LIN {X 0.120,Y -301.447,Z 452.705,A 0.000,B 0.000,C 90.000,E1 126.870} C_DIS
LIN {X -0.059,Y -305.207,Z 452.702,A 0.000,B 0.000,C 90.000,E1 126.423} C_DIS
LIN {X -0.045,Y -307.018,Z 452.700,A 0.000,B 0.000,C 90.000,E1 126.091} C_DIS
LIN {X 0.151,Y -308.441,Z 452.699,A 0.000,B 0.000,C 90.000,E1 125.724} C_DIS
LIN {X 0.025,Y -313.580,Z 452.690,A 0.000,B 0.000,C 90.000,E1 124.119} C_DIS
LIN {X 0.115,Y -323.537,Z 452.673,A 0.000,B 0.000,C 90.000,E1 121.209} C_DIS
LIN {X 0.173,Y -334.816,Z 452.658,A 0.000,B 0.000,C 90.000,E1 118.359} C_DIS
LIN {X 0.070,Y -347.524,Z 452.642,A 0.000,B 0.000,C 90.000,E1 115.591} C_DIS
LIN {X -0.180,Y -360.110,Z 452.629,A 0.000,B 0.000,C 90.000,E1 113.206} C_DIS
LIN {X 0.078,Y -374.006,Z 452.616,A 0.000,B 0.000,C 90.000,E1 110.791} C_DIS
LIN {X -0.054,Y -389.312,Z 452.603,A 0.000,B 0.000,C 90.000,E1 108.489} C_DIS
LIN {X 0.080,Y -406.143,Z 452.590,A 0.000,B 0.000,C 90.000,E1 106.205} C_DIS
LIN {X 0.012,Y -424.621,Z 452.578,A 0.000,B 0.000,C 90.000,E1 104.008} C_DIS
LIN {X 0.142,Y -444.522,Z 452.566,A 0.000,B 0.000,C 90.000,E1 101.883} C_DIS
LIN {X 0.031,Y -465.029,Z 452.555,A 0.000,B 0.000,C 90.000,E1 99.962} C_DIS
LIN {X 0.056,Y -483.349,Z 452.547,A 0.000,B 0.000,C 90.000,E1 98.398} C_DIS
LIN {X 0.226,Y -485.471,Z 452.546,A 0.000,B 0.000,C 90.000,E1 98.163} C_DIS
LIN {X 0.064,Y -487.300,Z 452.544,A 0.000,B 0.000,C 90.000,E1 97.936} C_DIS
LIN {X -0.032,Y -488.676,Z 452.543,A 0.000,B 0.000,C 90.000,E1 97.701} C_DIS
LIN {X 0.176,Y -490.427,Z 452.540,A 0.000,B 0.000,C 90.000,E1 97.182} C_DIS
LIN {X -0.095,Y -491.085,Z 452.537,A 0.000,B 0.000,C 90.000,E1 96.720} C_DIS
LIN {X 0.132,Y -490.756,Z 452.535,A 0.000,B 0.000,C 90.000,E1 96.201} C_DIS
LIN {X -0.126,Y -489.389,Z 452.532,A 0.000,B 0.000,C 90.000,E1 95.739} C_DIS
LIN {X 0.208,Y -488.246,Z 452.530,A 0.000,B 0.000,C 90.000,E1 95.454} C_DIS
LIN {X 0.100,Y -486.714,Z 452.529,A 0.000,B 0.000,C 90.000,E1 95.220} C_DIS
LIN {X -0.023,Y -478.801,Z 452.524,A 0.000,B 0.000,C 90.000,E1 94.245} C_DIS
LIN {X -0.206,Y -457.268,Z 452.508,A 0.000,B 0.000,C 90.000,E1 91.489} C_DIS
LIN {X -0.024,Y -444.971,Z 452.498,A 0.000,B 0.000,C 90.000,E1 89.656} C_DIS
LIN {X -0.084,Y -433.386,Z 452.488,A 0.000,B 0.000,C 90.000,E1 87.822} C_DIS
LIN {X -0.117,Y -418.721,Z 452.474,A 0.000,B 0.000,C 90.000,E1 85.412} C_DIS
LIN {X -0.119,Y -406.257,Z 452.462,A 0.000,B 0.000,C 90.000,E1 83.223} C_DIS
LIN {X 0.015,Y -395.531,Z 452.451,A 0.000,B 0.000,C 90.000,E1 81.254} C_DIS
LIN {X -0.039,Y -383.227,Z 452.439,A 0.000,B 0.000,C 90.000,E1 78.993} C_DIS
LIN {X -0.169,Y -368.243,Z 452.423,A 0.000,B 0.000,C 90.000,E1 76.117} C_DIS
LIN {X -0.106,Y -356.985,Z 452.410,A 0.000,B 0.000,C 90.000,E1 73.740} C_DIS
LIN {X -0.151,Y -342.943,Z 452.391,A 0.000,B 0.000,C 90.000,E1 70.423} C_DIS
LIN {X 0.038,Y -332.368,Z 452.376,A 0.000,B 0.000,C 90.000,E1 67.614} C_DIS
LIN {X 0.001,Y -321.989,Z 452.360,A 0.000,B 0.000,C 90.000,E1 64.793} C_DIS
LIN {X 0.035,Y -313.043,Z 452.346,A 0.000,B 0.000,C 90.000,E1 62.231} C_DIS
LIN {X -0.129,Y -304.242,Z 452.331,A 0.000,B 0.000,C 90.000,E1 59.665} C_DIS
LIN {X 0.016,Y -293.773,Z 452.313,A 0.000,B 0.000,C 90.000,E1 56.342} C_DIS
LIN {X 0.083,Y -284.083,Z 452.294,A 0.000,B 0.000,C 90.000,E1 52.970} C_DIS
LIN {X -0.107,Y -278.413,Z 452.283,A 0.000,B 0.000,C 90.000,E1 50.964} C_DIS
LIN {X 0.119,Y -272.507,Z 452.272,A 0.000,B 0.000,C 90.000,E1 48.852} C_DIS
LIN {X 0.026,Y -266.367,Z 452.260,A 0.000,B 0.000,C 90.000,E1 46.782} C_DIS
LIN {X -0.007,Y -260.067,Z 452.248,A 0.000,B 0.000,C 90.000,E1 44.676} C_DIS
LIN {X 0.030,Y -253.666,Z 452.236,A 0.000,B 0.000,C 90.000,E1 42.528} C_DIS
LIN {X -0.018,Y -245.018,Z 452.220,A 0.000,B 0.000,C 90.000,E1 39.644} C_DIS
LIN {X 0.084,Y -234.685,Z 452.200,A 0.000,B 0.000,C 90.000,E1 35.931} C_DIS
LIN {X -0.057,Y -227.197,Z 452.183,A 0.000,B 0.000,C 90.000,E1 32.959} C_DIS
LIN {X 0.072,Y -220.483,Z 452.166,A 0.000,B 0.000,C 90.000,E1 29.873} C_DIS
LIN {X 0.003,Y -214.671,Z 452.149,A 0.000,B 0.000,C 90.000,E1 26.796} C_DIS
LIN {X -0.085,Y -208.369,Z 452.127,A 0.000,B 0.000,C 90.000,E1 22.898} C_DIS
LIN {X -0.020,Y -203.087,Z 452.105,A 0.000,B 0.000,C 90.000,E1 18.906} C_DIS
LIN {X -0.056,Y -198.758,Z 452.083,A 0.000,B 0.000,C 90.000,E1 14.898} C_DIS
LIN {X -0.018,Y -194.835,Z 452.056,A 0.000,B 0.000,C 90.000,E1 10.018} C_DIS
LIN {X -0.064,Y -191.927,Z 452.024,A 0.000,B 0.000,C 90.000,E1 4.302} C_DIS
LIN {X 0.083,Y -191.956,Z 451.965,A 0.000,B 0.000,C 90.000,E1 353.742} C_DIS
LIN {X 0.097,Y -194.918,Z 451.933,A 0.000,B 0.000,C 90.000,E1 347.993} C_DIS
LIN {X -0.034,Y -198.884,Z 451.906,A 0.000,B 0.000,C 90.000,E1 343.142} C_DIS
LIN {X 0.035,Y -203.206,Z 451.884,A 0.000,B 0.000,C 90.000,E1 339.082} C_DIS
LIN {X -0.034,Y -208.624,Z 451.862,A 0.000,B 0.000,C 90.000,E1 335.101} C_DIS
LIN {X 0.041,Y -214.800,Z 451.840,A 0.000,B 0.000,C 90.000,E1 331.129} C_DIS
LIN {X -0.027,Y -221.542,Z 451.818,A 0.000,B 0.000,C 90.000,E1 327.248} C_DIS
LIN {X -0.075,Y -228.974,Z 451.797,A 0.000,B 0.000,C 90.000,E1 323.417} C_DIS
LIN {X -0.031,Y -237.180,Z 451.776,A 0.000,B 0.000,C 90.000,E1 319.622} C_DIS
LIN {X 0.023,Y -246.445,Z 451.755,A 0.000,B 0.000,C 90.000,E1 315.891} C_DIS
LIN {X 0.032,Y -256.044,Z 451.737,A 0.000,B 0.000,C 90.000,E1 312.609} C_DIS
LIN {X 0.055,Y -268.123,Z 451.717,A 0.000,B 0.000,C 90.000,E1 309.036} C_DIS
LIN {X 0.111,Y -280.070,Z 451.699,A 0.000,B 0.000,C 90.000,E1 305.884} C_DIS
LIN {X 0.018,Y -294.154,Z 451.681,A 0.000,B 0.000,C 90.000,E1 302.498} C_DIS
LIN {X -0.144,Y -307.643,Z 451.664,A 0.000,B 0.000,C 90.000,E1 299.539} C_DIS
LIN {X -0.045,Y -320.638,Z 451.650,A 0.000,B 0.000,C 90.000,E1 296.924} C_DIS
LIN {X -0.046,Y -334.871,Z 451.635,A 0.000,B 0.000,C 90.000,E1 294.387} C_DIS
LIN {X 0.021,Y -346.380,Z 451.625,A 0.000,B 0.000,C 90.000,E1 292.514} C_DIS
LIN {X -0.181,Y -363.228,Z 451.612,A 0.000,B 0.000,C 90.000,E1 290.120} C_DIS
LIN {X 0.035,Y -386.462,Z 451.595,A 0.000,B 0.000,C 90.000,E1 287.149} C_DIS
LIN {X -0.172,Y -401.479,Z 451.586,A 0.000,B 0.000,C 90.000,E1 285.481} C_DIS
LIN {X 0.187,Y -424.373,Z 451.573,A 0.000,B 0.000,C 90.000,E1 283.119} C_DIS
LIN {X 0.111,Y -434.478,Z 451.567,A 0.000,B 0.000,C 90.000,E1 282.119} C_DIS
LIN {X -0.239,Y -444.292,Z 451.562,A 0.000,B 0.000,C 90.000,E1 281.130} C_DIS
LIN {X 0.076,Y -451.255,Z 451.557,A 0.000,B 0.000,C 90.000,E1 280.310} C_DIS
LIN {X -0.146,Y -457.806,Z 451.553,A 0.000,B 0.000,C 90.000,E1 279.557} C_DIS
LIN {X 0.151,Y -463.921,Z 451.549,A 0.000,B 0.000,C 90.000,E1 278.746} C_DIS
LIN {X 0.043,Y -469.402,Z 451.544,A 0.000,B 0.000,C 90.000,E1 277.992} C_DIS
LIN {X -0.017,Y -474.376,Z 451.540,A 0.000,B 0.000,C 90.000,E1 277.239} C_DIS
LIN {X -0.234,Y -480.245,Z 451.535,A 0.000,B 0.000,C 90.000,E1 276.258} C_DIS
LIN {X -0.261,Y -484.098,Z 451.530,A 0.000,B 0.000,C 90.000,E1 275.511} C_DIS
LIN {X -0.080,Y -486.395,Z 451.528,A 0.000,B 0.000,C 90.000,E1 274.992} C_DIS
LIN {X 0.114,Y -488.309,Z 451.525,A 0.000,B 0.000,C 90.000,E1 274.473} C_DIS
LIN {X -0.176,Y -489.851,Z 451.522,A 0.000,B 0.000,C 90.000,E1 274.012} C_DIS
LIN {X 0.001,Y -490.957,Z 451.519,A 0.000,B 0.000,C 90.000,E1 273.498} C_DIS
LIN {X 0.216,Y -491.675,Z 451.517,A 0.000,B 0.000,C 90.000,E1 272.980} C_DIS
LIN {X -0.079,Y -492.019,Z 451.514,A 0.000,B 0.000,C 90.000,E1 272.522} C_DIS
LIN {X 0.125,Y -491.944,Z 451.511,A 0.000,B 0.000,C 90.000,E1 272.007} C_DIS
LIN {X -0.144,Y -491.479,Z 451.508,A 0.000,B 0.000,C 90.000,E1 271.547} C_DIS
LIN {X 0.060,Y -490.612,Z 451.506,A 0.000,B 0.000,C 90.000,E1 271.031} C_DIS
LIN {X -0.225,Y -489.255,Z 451.503,A 0.000,B 0.000,C 90.000,E1 270.573} C_DIS
LIN {X -0.026,Y -487.379,Z 451.500,A 0.000,B 0.000,C 90.000,E1 270.057} C_DIS
LIN {X 0.164,Y -484.887,Z 451.498,A 0.000,B 0.000,C 90.000,E1 269.542} C_DIS
LIN {X -0.148,Y -481.651,Z 451.495,A 0.000,B 0.000,C 90.000,E1 269.083} C_DIS
LIN {X 0.005,Y -477.481,Z 451.492,A 0.000,B 0.000,C 90.000,E1 268.568} C_DIS
LIN {X -0.167,Y -475.019,Z 451.491,A 0.000,B 0.000,C 90.000,E1 268.339} C_DIS
LIN {X 0.129,Y -469.421,Z 451.488,A 0.000,B 0.000,C 90.000,E1 267.822} C_DIS
LIN {X -0.119,Y -463.170,Z 451.486,A 0.000,B 0.000,C 90.000,E1 267.421} C_DIS
LIN {X 0.143,Y -456.577,Z 451.484,A 0.000,B 0.000,C 90.000,E1 267.020} C_DIS
LIN {X -0.034,Y -449.739,Z 451.482,A 0.000,B 0.000,C 90.000,E1 266.731} C_DIS
LIN {X 0.132,Y -442.560,Z 451.480,A 0.000,B 0.000,C 90.000,E1 266.445} C_DIS
LIN {X -0.190,Y -434.851,Z 451.479,A 0.000,B 0.000,C 90.000,E1 266.274} C_DIS
LIN {X -0.091,Y -426.271,Z 451.478,A 0.000,B 0.000,C 90.000,E1 266.102} C_DIS
LIN {X -0.040,Y -414.893,Z 451.478,A 0.000,B 0.000,C 90.000,E1 265.988} C_DIS
LIN {X 0.146,Y -408.689,Z 451.478,A 0.000,B 0.000,C 90.000,E1 265.931} C_DIS
LIN {X 0.044,Y -180.918,Z 451.477,A 0.000,B 0.000,C 90.000,E1 265.927} C_DIS
LIN {X 0.076,Y -180.841,Z 451.472,A 0.000,B 0.000,C 90.000,E1 264.894} C_DIS
LIN {X -0.027,Y -178.883,Z 451.443,A 0.000,B 0.000,C 90.000,E1 259.690} C_DIS
LIN {X 0.048,Y -175.926,Z 451.414,A 0.000,B 0.000,C 90.000,E1 254.574} C_DIS
LIN {X -0.006,Y -175.365,Z 451.410,A 0.000,B 0.000,C 90.000,E1 253.740} C_DIS
LIN {X 0.052,Y -172.143,Z 451.386,A 0.000,B 0.000,C 90.000,E1 249.444} C_DIS
LIN {X 0.029,Y -171.608,Z 451.381,A 0.000,B 0.000,C 90.000,E1 248.592} C_DIS
LIN {X 0.018,Y -167.830,Z 451.357,A 0.000,B 0.000,C 90.000,E1 244.280} C_DIS
LIN {X 0.035,Y -166.556,Z 451.348,A 0.000,B 0.000,C 90.000,E1 242.538} C_DIS
LIN {X -0.054,Y -162.551,Z 451.323,A 0.000,B 0.000,C 90.000,E1 238.201} C_DIS
LIN {X 0.005,Y -161.229,Z 451.313,A 0.000,B 0.000,C 90.000,E1 236.421} C_DIS
LIN {X 0.041,Y -157.234,Z 451.289,A 0.000,B 0.000,C 90.000,E1 231.984} C_DIS
LIN {X 0.064,Y -155.959,Z 451.279,A 0.000,B 0.000,C 90.000,E1 230.194} C_DIS
LIN {X 0.021,Y -152.213,Z 451.254,A 0.000,B 0.000,C 90.000,E1 225.729} C_DIS
LIN {X 0.042,Y -150.457,Z 451.239,A 0.000,B 0.000,C 90.000,E1 223.014} C_DIS
LIN {X 0.069,Y -147.183,Z 451.214,A 0.000,B 0.000,C 90.000,E1 218.463} C_DIS
LIN {X 0.035,Y -145.201,Z 451.194,A 0.000,B 0.000,C 90.000,E1 214.818} C_DIS
LIN {X -0.055,Y -142.338,Z 451.163,A 0.000,B 0.000,C 90.000,E1 209.333} C_DIS
LIN {X -0.001,Y -141.727,Z 451.153,A 0.000,B 0.000,C 90.000,E1 207.462} C_DIS
LIN {X -0.019,Y -139.480,Z 451.116,A 0.000,B 0.000,C 90.000,E1 200.972} C_DIS
LIN {X -0.030,Y -138.979,Z 451.101,A 0.000,B 0.000,C 90.000,E1 198.181} C_DIS
LIN {X -0.045,Y -138.332,Z 451.054,A 0.000,B 0.000,C 90.000,E1 189.782} C_DIS
LIN {X -0.045,Y -139.429,Z 451.008,A 0.000,B 0.000,C 90.000,E1 181.375} C_DIS
LIN {X 0.008,Y -141.357,Z 450.971,A 0.000,B 0.000,C 90.000,E1 174.837} C_DIS
LIN {X -0.016,Y -142.711,Z 450.956,A 0.000,B 0.000,C 90.000,E1 172.064} C_DIS
LIN {X -0.056,Y -145.086,Z 450.930,A 0.000,B 0.000,C 90.000,E1 167.465} C_DIS
LIN {X -0.061,Y -147.710,Z 450.910,A 0.000,B 0.000,C 90.000,E1 163.795} C_DIS
LIN {X 0.022,Y -150.365,Z 450.890,A 0.000,B 0.000,C 90.000,E1 160.115} C_DIS
LIN {X 0.041,Y -153.792,Z 450.869,A 0.000,B 0.000,C 90.000,E1 156.485} C_DIS
LIN {X -0.039,Y -157.204,Z 450.849,A 0.000,B 0.000,C 90.000,E1 152.922} C_DIS
LIN {X 0.042,Y -161.366,Z 450.830,A 0.000,B 0.000,C 90.000,E1 149.331} C_DIS
LIN {X 0.053,Y -165.569,Z 450.810,A 0.000,B 0.000,C 90.000,E1 145.801} C_DIS
LIN {X -0.063,Y -170.486,Z 450.791,A 0.000,B 0.000,C 90.000,E1 142.351} C_DIS
LIN {X 0.086,Y -175.368,Z 450.772,A 0.000,B 0.000,C 90.000,E1 138.852} C_DIS
LIN {X -0.051,Y -180.991,Z 450.753,A 0.000,B 0.000,C 90.000,E1 135.486} C_DIS
LIN {X 0.073,Y -186.418,Z 450.734,A 0.000,B 0.000,C 90.000,E1 132.081} C_DIS
LIN {X -0.126,Y -191.046,Z 450.720,A 0.000,B 0.000,C 90.000,E1 129.644} C_DIS
LIN {X 0.003,Y -195.023,Z 450.707,A 0.000,B 0.000,C 90.000,E1 127.282} C_DIS
LIN {X -0.030,Y -292.656,Z 450.707,A 0.000,B 0.000,C 90.000,E1 127.282} C_DIS
LIN {X -0.113,Y -297.600,Z 450.706,A 0.000,B 0.000,C 90.000,E1 127.156} C_DIS
LIN {X 0.008,Y -300.299,Z 450.705,A 0.000,B 0.000,C 90.000,E1 126.950} C_DIS
LIN {X 0.027,Y -304.083,Z 450.703,A 0.000,B 0.000,C 90.000,E1 126.537} C_DIS
LIN {X 0.135,Y -306.022,Z 450.701,A 0.000,B 0.000,C 90.000,E1 126.217} C_DIS
LIN {X 0.059,Y -307.557,Z 450.700,A 0.000,B 0.000,C 90.000,E1 125.931} C_DIS
LIN {X 0.090,Y -308.890,Z 450.698,A 0.000,B 0.000,C 90.000,E1 125.598} C_DIS
LIN {X -0.005,Y -320.535,Z 450.678,A 0.000,B 0.000,C 90.000,E1 122.054} C_DIS
LIN {X -0.048,Y -331.424,Z 450.662,A 0.000,B 0.000,C 90.000,E1 119.205} C_DIS
LIN {X -0.103,Y -343.712,Z 450.647,A 0.000,B 0.000,C 90.000,E1 116.411} C_DIS
LIN {X 0.013,Y -355.896,Z 450.633,A 0.000,B 0.000,C 90.000,E1 113.951} C_DIS
LIN {X 0.168,Y -369.359,Z 450.620,A 0.000,B 0.000,C 90.000,E1 111.535} C_DIS
LIN {X 0.055,Y -384.199,Z 450.607,A 0.000,B 0.000,C 90.000,E1 109.214} C_DIS
LIN {X 0.181,Y -400.526,Z 450.594,A 0.000,B 0.000,C 90.000,E1 106.913} C_DIS
LIN {X -0.028,Y -418.459,Z 450.582,A 0.000,B 0.000,C 90.000,E1 104.717} C_DIS
LIN {X 0.194,Y -438.015,Z 450.570,A 0.000,B 0.000,C 90.000,E1 102.535} C_DIS
LIN {X 0.191,Y -458.346,Z 450.559,A 0.000,B 0.000,C 90.000,E1 100.546} C_DIS
LIN {X -0.250,Y -484.346,Z 450.546,A 0.000,B 0.000,C 90.000,E1 98.341} C_DIS
LIN {X -0.039,Y -487.846,Z 450.544,A 0.000,B 0.000,C 90.000,E1 97.871} C_DIS
LIN {X -0.220,Y -489.138,Z 450.542,A 0.000,B 0.000,C 90.000,E1 97.644} C_DIS
LIN {X 0.150,Y -490.088,Z 450.541,A 0.000,B 0.000,C 90.000,E1 97.352} C_DIS
LIN {X -0.120,Y -491.128,Z 450.538,A 0.000,B 0.000,C 90.000,E1 96.891} C_DIS
LIN {X 0.103,Y -491.164,Z 450.535,A 0.000,B 0.000,C 90.000,E1 96.372} C_DIS
LIN {X -0.155,Y -490.200,Z 450.533,A 0.000,B 0.000,C 90.000,E1 95.910} C_DIS
LIN {X 0.072,Y -488.065,Z 450.530,A 0.000,B 0.000,C 90.000,E1 95.391} C_DIS
LIN {X -0.082,Y -486.413,Z 450.529,A 0.000,B 0.000,C 90.000,E1 95.163} C_DIS
LIN {X 0.137,Y -476.456,Z 450.522,A 0.000,B 0.000,C 90.000,E1 93.898} C_DIS
LIN {X 0.076,Y -456.937,Z 450.508,A 0.000,B 0.000,C 90.000,E1 91.375} C_DIS
LIN {X -0.206,Y -444.676,Z 450.498,A 0.000,B 0.000,C 90.000,E1 89.599} C_DIS
LIN {X 0.170,Y -433.088,Z 450.487,A 0.000,B 0.000,C 90.000,E1 87.707} C_DIS
LIN {X 0.114,Y -418.435,Z 450.474,A 0.000,B 0.000,C 90.000,E1 85.298} C_DIS
LIN {X 0.200,Y -404.474,Z 450.460,A 0.000,B 0.000,C 90.000,E1 82.818} C_DIS
LIN {X -0.100,Y -393.730,Z 450.449,A 0.000,B 0.000,C 90.000,E1 80.905} C_DIS
LIN {X -0.154,Y -383.001,Z 450.438,A 0.000,B 0.000,C 90.000,E1 78.926} C_DIS
LIN {X 0.085,Y -368.056,Z 450.422,A 0.000,B 0.000,C 90.000,E1 75.992} C_DIS
LIN {X 0.089,Y -355.495,Z 450.407,A 0.000,B 0.000,C 90.000,E1 73.323} C_DIS
LIN {X -0.017,Y -341.580,Z 450.389,A 0.000,B 0.000,C 90.000,E1 70.007} C_DIS
LIN {X -0.057,Y -331.015,Z 450.373,A 0.000,B 0.000,C 90.000,E1 67.230} C_DIS
LIN {X -0.123,Y -320.640,Z 450.358,A 0.000,B 0.000,C 90.000,E1 64.409} C_DIS
LIN {X -0.120,Y -311.662,Z 450.343,A 0.000,B 0.000,C 90.000,E1 61.847} C_DIS
LIN {X 0.100,Y -302.879,Z 450.329,A 0.000,B 0.000,C 90.000,E1 59.203} C_DIS
LIN {X -0.053,Y -292.500,Z 450.311,A 0.000,B 0.000,C 90.000,E1 55.928} C_DIS
LIN {X -0.027,Y -282.862,Z 450.292,A 0.000,B 0.000,C 90.000,E1 52.557} C_DIS
LIN {X -0.068,Y -277.160,Z 450.281,A 0.000,B 0.000,C 90.000,E1 50.517} C_DIS
LIN {X 0.133,Y -271.205,Z 450.269,A 0.000,B 0.000,C 90.000,E1 48.405} C_DIS
LIN {X 0.002,Y -265.041,Z 450.257,A 0.000,B 0.000,C 90.000,E1 46.338} C_DIS
LIN {X 0.134,Y -258.725,Z 450.246,A 0.000,B 0.000,C 90.000,E1 44.190} C_DIS
LIN {X -0.028,Y -252.292,Z 450.234,A 0.000,B 0.000,C 90.000,E1 42.081} C_DIS
LIN {X -0.106,Y -243.674,Z 450.218,A 0.000,B 0.000,C 90.000,E1 39.197} C_DIS
LIN {X 0.008,Y -233.449,Z 450.197,A 0.000,B 0.000,C 90.000,E1 35.471} C_DIS
LIN {X -0.032,Y -226.071,Z 450.180,A 0.000,B 0.000,C 90.000,E1 32.467} C_DIS
LIN {X -0.046,Y -219.536,Z 450.163,A 0.000,B 0.000,C 90.000,E1 29.411} C_DIS
LIN {X 0.053,Y -213.838,Z 450.146,A 0.000,B 0.000,C 90.000,E1 26.283} C_DIS
LIN {X -0.064,Y -207.639,Z 450.124,A 0.000,B 0.000,C 90.000,E1 22.386} C_DIS
LIN {X 0.092,Y -202.488,Z 450.102,A 0.000,B 0.000,C 90.000,E1 18.362} C_DIS
LIN {X 0.032,Y -198.234,Z 450.080,A 0.000,B 0.000,C 90.000,E1 14.356} C_DIS
LIN {X -0.033,Y -194.424,Z 450.053,A 0.000,B 0.000,C 90.000,E1 9.500} C_DIS
LIN {X -0.092,Y -191.658,Z 450.021,A 0.000,B 0.000,C 90.000,E1 3.784} C_DIS
LIN {X 0.078,Y -191.838,Z 449.965,A 0.000,B 0.000,C 90.000,E1 353.742} C_DIS
LIN {X 0.086,Y -194.788,Z 449.933,A 0.000,B 0.000,C 90.000,E1 347.993} C_DIS
LIN {X -0.050,Y -198.736,Z 449.906,A 0.000,B 0.000,C 90.000,E1 343.142} C_DIS
LIN {X 0.014,Y -203.042,Z 449.884,A 0.000,B 0.000,C 90.000,E1 339.082} C_DIS
LIN {X -0.060,Y -208.464,Z 449.862,A 0.000,B 0.000,C 90.000,E1 335.101} C_DIS
LIN {X 0.008,Y -214.633,Z 449.840,A 0.000,B 0.000,C 90.000,E1 331.129} C_DIS
LIN {X -0.066,Y -221.378,Z 449.818,A 0.000,B 0.000,C 90.000,E1 327.248} C_DIS
LIN {X -0.120,Y -228.829,Z 449.797,A 0.000,B 0.000,C 90.000,E1 323.417} C_DIS
LIN {X -0.083,Y -237.051,Z 449.776,A 0.000,B 0.000,C 90.000,E1 319.622} C_DIS
LIN {X 0.006,Y -244.340,Z 449.759,A 0.000,B 0.000,C 90.000,E1 316.620} C_DIS
LIN {X -0.055,Y -253.675,Z 449.741,A 0.000,B 0.000,C 90.000,E1 313.338} C_DIS
LIN {X 0.011,Y -264.316,Z 449.723,A 0.000,B 0.000,C 90.000,E1 310.092} C_DIS
LIN {X -0.093,Y -275.906,Z 449.705,A 0.000,B 0.000,C 90.000,E1 306.950} C_DIS
LIN {X 0.021,Y -288.375,Z 449.688,A 0.000,B 0.000,C 90.000,E1 303.833} C_DIS
LIN {X 0.101,Y -301.526,Z 449.671,A 0.000,B 0.000,C 90.000,E1 300.797} C_DIS
LIN {X 0.168,Y -317.259,Z 449.653,A 0.000,B 0.000,C 90.000,E1 297.513} C_DIS
LIN {X 0.195,Y -333.045,Z 449.637,A 0.000,B 0.000,C 90.000,E1 294.643} C_DIS
LIN {X -0.081,Y -344.418,Z 449.627,A 0.000,B 0.000,C 90.000,E1 292.823} C_DIS
LIN {X 0.001,Y -361.085,Z 449.613,A 0.000,B 0.000,C 90.000,E1 290.375} C_DIS
LIN {X -0.068,Y -386.502,Z 449.595,A 0.000,B 0.000,C 90.000,E1 287.149} C_DIS
LIN {X 0.146,Y -401.533,Z 449.586,A 0.000,B 0.000,C 90.000,E1 285.426} C_DIS
LIN {X 0.053,Y -424.602,Z 449.573,A 0.000,B 0.000,C 90.000,E1 283.119} C_DIS
LIN {X -0.021,Y -434.708,Z 449.567,A 0.000,B 0.000,C 90.000,E1 282.119} C_DIS
LIN {X 0.043,Y -444.532,Z 449.562,A 0.000,B 0.000,C 90.000,E1 281.074} C_DIS
LIN {X -0.124,Y -451.518,Z 449.557,A 0.000,B 0.000,C 90.000,E1 280.310} C_DIS
LIN {X -0.077,Y -460.132,Z 449.551,A 0.000,B 0.000,C 90.000,E1 279.265} C_DIS
LIN {X -0.224,Y -466.022,Z 449.547,A 0.000,B 0.000,C 90.000,E1 278.511} C_DIS
LIN {X -0.008,Y -472.957,Z 449.541,A 0.000,B 0.000,C 90.000,E1 277.466} C_DIS
LIN {X 0.231,Y -479.014,Z 449.536,A 0.000,B 0.000,C 90.000,E1 276.429} C_DIS
LIN {X 0.019,Y -484.258,Z 449.530,A 0.000,B 0.000,C 90.000,E1 275.454} C_DIS
LIN {X 0.202,Y -486.532,Z 449.528,A 0.000,B 0.000,C 90.000,E1 274.935} C_DIS
LIN {X -0.088,Y -488.459,Z 449.525,A 0.000,B 0.000,C 90.000,E1 274.473} C_DIS
LIN {X 0.111,Y -489.980,Z 449.522,A 0.000,B 0.000,C 90.000,E1 273.955} C_DIS
LIN {X -0.201,Y -491.048,Z 449.519,A 0.000,B 0.000,C 90.000,E1 273.498} C_DIS
LIN {X 0.015,Y -491.747,Z 449.517,A 0.000,B 0.000,C 90.000,E1 272.980} C_DIS
LIN {X 0.212,Y -492.036,Z 449.514,A 0.000,B 0.000,C 90.000,E1 272.465} C_DIS
LIN {X -0.075,Y -491.945,Z 449.511,A 0.000,B 0.000,C 90.000,E1 272.007} C_DIS
LIN {X 0.146,Y -491.465,Z 449.508,A 0.000,B 0.000,C 90.000,E1 271.489} C_DIS
LIN {X -0.139,Y -490.569,Z 449.506,A 0.000,B 0.000,C 90.000,E1 271.031} C_DIS
LIN {X 0.064,Y -489.232,Z 449.503,A 0.000,B 0.000,C 90.000,E1 270.516} C_DIS
LIN {X -0.225,Y -487.297,Z 449.500,A 0.000,B 0.000,C 90.000,E1 270.057} C_DIS
LIN {X 0.114,Y -486.154,Z 449.499,A 0.000,B 0.000,C 90.000,E1 269.771} C_DIS
LIN {X -0.190,Y -483.272,Z 449.496,A 0.000,B 0.000,C 90.000,E1 269.312} C_DIS
LIN {X 0.136,Y -481.554,Z 449.495,A 0.000,B 0.000,C 90.000,E1 269.026} C_DIS
LIN {X -0.190,Y -477.345,Z 449.492,A 0.000,B 0.000,C 90.000,E1 268.568} C_DIS
LIN {X 0.113,Y -474.872,Z 449.491,A 0.000,B 0.000,C 90.000,E1 268.282} C_DIS
LIN {X -0.039,Y -469.229,Z 449.488,A 0.000,B 0.000,C 90.000,E1 267.822} C_DIS
LIN {X -0.034,Y -466.123,Z 449.487,A 0.000,B 0.000,C 90.000,E1 267.593} C_DIS
LIN {X -0.056,Y -459.482,Z 449.484,A 0.000,B 0.000,C 90.000,E1 267.192} C_DIS
LIN {X 0.051,Y -452.770,Z 449.483,A 0.000,B 0.000,C 90.000,E1 266.846} C_DIS
LIN {X 0.092,Y -445.852,Z 449.481,A 0.000,B 0.000,C 90.000,E1 266.560} C_DIS
LIN {X 0.009,Y -438.228,Z 449.480,A 0.000,B 0.000,C 90.000,E1 266.331} C_DIS
LIN {X -0.089,Y -430.052,Z 449.479,A 0.000,B 0.000,C 90.000,E1 266.159} C_DIS
LIN {X -0.198,Y -419.921,Z 449.478,A 0.000,B 0.000,C 90.000,E1 266.045} C_DIS
LIN {X 0.184,Y -410.098,Z 449.478,A 0.000,B 0.000,C 90.000,E1 265.931} C_DIS
LIN {X 0.139,Y -406.147,Z 449.477,A 0.000,B 0.000,C 90.000,E1 265.927} C_DIS
LIN {X 0.029,Y -180.918,Z 449.477,A 0.000,B 0.000,C 90.000,E1 265.927} C_DIS
LIN {X 0.061,Y -180.840,Z 449.472,A 0.000,B 0.000,C 90.000,E1 264.894} C_DIS
LIN {X -0.042,Y -178.882,Z 449.443,A 0.000,B 0.000,C 90.000,E1 259.690} C_DIS
LIN {X 0.034,Y -175.924,Z 449.414,A 0.000,B 0.000,C 90.000,E1 254.574} C_DIS
LIN {X -0.021,Y -175.361,Z 449.410,A 0.000,B 0.000,C 90.000,E1 253.740} C_DIS
LIN {X 0.038,Y -172.141,Z 449.386,A 0.000,B 0.000,C 90.000,E1 249.444} C_DIS
LIN {X 0.015,Y -171.604,Z 449.381,A 0.000,B 0.000,C 90.000,E1 248.592} C_DIS
LIN {X 0.004,Y -167.827,Z 449.357,A 0.000,B 0.000,C 90.000,E1 244.280} C_DIS
LIN {X 0.021,Y -166.551,Z 449.347,A 0.000,B 0.000,C 90.000,E1 242.538} C_DIS
LIN {X -0.069,Y -162.547,Z 449.323,A 0.000,B 0.000,C 90.000,E1 238.201} C_DIS
LIN {X -0.009,Y -161.225,Z 449.313,A 0.000,B 0.000,C 90.000,E1 236.421} C_DIS
LIN {X 0.027,Y -157.231,Z 449.289,A 0.000,B 0.000,C 90.000,E1 231.984} C_DIS
LIN {X 0.050,Y -155.955,Z 449.279,A 0.000,B 0.000,C 90.000,E1 230.194} C_DIS
LIN {X 0.008,Y -152.209,Z 449.254,A 0.000,B 0.000,C 90.000,E1 225.729} C_DIS
LIN {X 0.029,Y -150.454,Z 449.239,A 0.000,B 0.000,C 90.000,E1 223.014} C_DIS
LIN {X 0.056,Y -147.180,Z 449.214,A 0.000,B 0.000,C 90.000,E1 218.463} C_DIS
LIN {X 0.022,Y -145.197,Z 449.193,A 0.000,B 0.000,C 90.000,E1 214.818} C_DIS
LIN {X 0.057,Y -142.336,Z 449.163,A 0.000,B 0.000,C 90.000,E1 209.283} C_DIS
LIN {X -0.014,Y -141.725,Z 449.153,A 0.000,B 0.000,C 90.000,E1 207.462} C_DIS
LIN {X -0.032,Y -139.479,Z 449.116,A 0.000,B 0.000,C 90.000,E1 200.972} C_DIS
LIN {X -0.043,Y -138.977,Z 449.101,A 0.000,B 0.000,C 90.000,E1 198.181} C_DIS
LIN {X 0.078,Y -138.331,Z 449.054,A 0.000,B 0.000,C 90.000,E1 189.726} C_DIS
LIN {X -0.058,Y -139.431,Z 449.008,A 0.000,B 0.000,C 90.000,E1 181.375} C_DIS
LIN {X 0.021,Y -140.956,Z 448.976,A 0.000,B 0.000,C 90.000,E1 175.755} C_DIS
LIN {X -0.029,Y -142.713,Z 448.956,A 0.000,B 0.000,C 90.000,E1 172.064} C_DIS
LIN {X 0.071,Y -145.089,Z 448.930,A 0.000,B 0.000,C 90.000,E1 167.409} C_DIS
LIN {X 0.068,Y -147.714,Z 448.910,A 0.000,B 0.000,C 90.000,E1 163.740} C_DIS
LIN {X 0.009,Y -150.370,Z 448.890,A 0.000,B 0.000,C 90.000,E1 160.115} C_DIS
LIN {X 0.026,Y -153.797,Z 448.869,A 0.000,B 0.000,C 90.000,E1 156.485} C_DIS
LIN {X 0.087,Y -157.209,Z 448.849,A 0.000,B 0.000,C 90.000,E1 152.871} C_DIS
LIN {X 0.028,Y -161.373,Z 448.830,A 0.000,B 0.000,C 90.000,E1 149.331} C_DIS
LIN {X 0.039,Y -165.575,Z 448.810,A 0.000,B 0.000,C 90.000,E1 145.801} C_DIS
LIN {X 0.027,Y -170.495,Z 448.791,A 0.000,B 0.000,C 90.000,E1 142.316} C_DIS
LIN {X 0.071,Y -175.375,Z 448.772,A 0.000,B 0.000,C 90.000,E1 138.852} C_DIS
LIN {X -0.066,Y -180.999,Z 448.753,A 0.000,B 0.000,C 90.000,E1 135.486} C_DIS
LIN {X 0.058,Y -186.427,Z 448.734,A 0.000,B 0.000,C 90.000,E1 132.081} C_DIS
LIN {X 0.006,Y -191.053,Z 448.720,A 0.000,B 0.000,C 90.000,E1 129.600} C_DIS
LIN {X -0.057,Y -195.139,Z 448.707,A 0.000,B 0.000,C 90.000,E1 127.237} C_DIS
LIN {X -0.120,Y -293.286,Z 448.707,A 0.000,B 0.000,C 90.000,E1 127.237} C_DIS
LIN {X -0.136,Y -296.587,Z 448.706,A 0.000,B 0.000,C 90.000,E1 127.156} C_DIS
LIN {X 0.085,Y -299.495,Z 448.705,A 0.000,B 0.000,C 90.000,E1 126.950} C_DIS
LIN {X -0.049,Y -303.164,Z 448.703,A 0.000,B 0.000,C 90.000,E1 126.629} C_DIS
LIN {X -0.058,Y -306.746,Z 448.700,A 0.000,B 0.000,C 90.000,E1 126.091} C_DIS
LIN {X 0.143,Y -308.289,Z 448.699,A 0.000,B 0.000,C 90.000,E1 125.724} C_DIS
LIN {X -0.086,Y -309.508,Z 448.697,A 0.000,B 0.000,C 90.000,E1 125.438} C_DIS
LIN {X -0.150,Y -320.047,Z 448.679,A 0.000,B 0.000,C 90.000,E1 122.212} C_DIS
LIN {X -0.038,Y -330.874,Z 448.663,A 0.000,B 0.000,C 90.000,E1 119.333} C_DIS
LIN {X -0.110,Y -343.095,Z 448.647,A 0.000,B 0.000,C 90.000,E1 116.539} C_DIS
LIN {X -0.009,Y -355.215,Z 448.634,A 0.000,B 0.000,C 90.000,E1 114.079} C_DIS
LIN {X 0.129,Y -368.610,Z 448.620,A 0.000,B 0.000,C 90.000,E1 111.663} C_DIS
LIN {X 0.127,Y -383.377,Z 448.607,A 0.000,B 0.000,C 90.000,E1 109.322} C_DIS
LIN {X 0.107,Y -399.624,Z 448.595,A 0.000,B 0.000,C 90.000,E1 107.040} C_DIS
LIN {X -0.014,Y -417.471,Z 448.582,A 0.000,B 0.000,C 90.000,E1 104.828} C_DIS
LIN {X 0.151,Y -436.966,Z 448.570,A 0.000,B 0.000,C 90.000,E1 102.647} C_DIS
LIN {X 0.067,Y -457.268,Z 448.559,A 0.000,B 0.000,C 90.000,E1 100.658} C_DIS
LIN {X -0.070,Y -480.720,Z 448.548,A 0.000,B 0.000,C 90.000,E1 98.624} C_DIS
LIN {X 0.008,Y -483.374,Z 448.547,A 0.000,B 0.000,C 90.000,E1 98.398} C_DIS
LIN {X 0.172,Y -485.583,Z 448.545,A 0.000,B 0.000,C 90.000,E1 98.163} C_DIS
LIN {X -0.214,Y -487.265,Z 448.544,A 0.000,B 0.000,C 90.000,E1 97.992} C_DIS
LIN {X 0.160,Y -488.744,Z 448.543,A 0.000,B 0.000,C 90.000,E1 97.701} C_DIS
LIN {X 0.047,Y -489.847,Z 448.542,A 0.000,B 0.000,C 90.000,E1 97.466} C_DIS
LIN {X 0.262,Y -491.145,Z 448.539,A 0.000,B 0.000,C 90.000,E1 96.947} C_DIS
LIN {X -0.004,Y -491.413,Z 448.536,A 0.000,B 0.000,C 90.000,E1 96.486} C_DIS
LIN {X 0.224,Y -490.693,Z 448.533,A 0.000,B 0.000,C 90.000,E1 95.967} C_DIS
LIN {X -0.082,Y -488.865,Z 448.531,A 0.000,B 0.000,C 90.000,E1 95.511} C_DIS
LIN {X -0.189,Y -487.424,Z 448.529,A 0.000,B 0.000,C 90.000,E1 95.277} C_DIS
LIN {X 0.177,Y -479.581,Z 448.524,A 0.000,B 0.000,C 90.000,E1 94.245} C_DIS
LIN {X -0.205,Y -456.102,Z 448.507,A 0.000,B 0.000,C 90.000,E1 91.260} C_DIS
LIN {X 0.143,Y -442.263,Z 448.495,A 0.000,B 0.000,C 90.000,E1 89.141} C_DIS
LIN {X 0.169,Y -429.034,Z 448.484,A 0.000,B 0.000,C 90.000,E1 87.020} C_DIS
LIN {X -0.168,Y -411.476,Z 448.467,A 0.000,B 0.000,C 90.000,E1 84.090} C_DIS
LIN {X 0.016,Y -400.728,Z 448.456,A 0.000,B 0.000,C 90.000,E1 82.129} C_DIS
LIN {X 0.028,Y -391.517,Z 448.447,A 0.000,B 0.000,C 90.000,E1 80.443} C_DIS
LIN {X -0.081,Y -380.839,Z 448.436,A 0.000,B 0.000,C 90.000,E1 78.465} C_DIS
LIN {X 0.089,Y -367.474,Z 448.421,A 0.000,B 0.000,C 90.000,E1 75.825} C_DIS
LIN {X 0.172,Y -354.978,Z 448.406,A 0.000,B 0.000,C 90.000,E1 73.142} C_DIS
LIN {X 0.052,Y -339.899,Z 448.386,A 0.000,B 0.000,C 90.000,E1 69.518} C_DIS
LIN {X -0.012,Y -330.500,Z 448.372,A 0.000,B 0.000,C 90.000,E1 67.050} C_DIS
LIN {X 0.037,Y -320.088,Z 448.357,A 0.000,B 0.000,C 90.000,E1 64.204} C_DIS
LIN {X 0.028,Y -311.100,Z 448.342,A 0.000,B 0.000,C 90.000,E1 61.641} C_DIS
LIN {X 0.202,Y -303.373,Z 448.330,A 0.000,B 0.000,C 90.000,E1 59.331} C_DIS
LIN {X -0.107,Y -292.933,Z 448.311,A 0.000,B 0.000,C 90.000,E1 56.087} C_DIS
LIN {X -0.073,Y -283.271,Z 448.293,A 0.000,B 0.000,C 90.000,E1 52.718} C_DIS
LIN {X 0.067,Y -277.578,Z 448.281,A 0.000,B 0.000,C 90.000,E1 50.642} C_DIS
LIN {X -0.105,Y -271.658,Z 448.270,A 0.000,B 0.000,C 90.000,E1 48.609} C_DIS
LIN {X -0.024,Y -265.518,Z 448.258,A 0.000,B 0.000,C 90.000,E1 46.500} C_DIS
LIN {X 0.118,Y -259.224,Z 448.247,A 0.000,B 0.000,C 90.000,E1 44.352} C_DIS
LIN {X -0.036,Y -252.792,Z 448.235,A 0.000,B 0.000,C 90.000,E1 42.243} C_DIS
LIN {X -0.098,Y -244.164,Z 448.219,A 0.000,B 0.000,C 90.000,E1 39.358} C_DIS
LIN {X -0.018,Y -233.907,Z 448.198,A 0.000,B 0.000,C 90.000,E1 35.644} C_DIS
LIN {X 0.013,Y -226.501,Z 448.181,A 0.000,B 0.000,C 90.000,E1 32.625} C_DIS
LIN {X -0.066,Y -219.928,Z 448.164,A 0.000,B 0.000,C 90.000,E1 29.589} C_DIS
LIN {X -0.059,Y -214.151,Z 448.147,A 0.000,B 0.000,C 90.000,E1 26.488} C_DIS
LIN {X 0.116,Y -207.905,Z 448.125,A 0.000,B 0.000,C 90.000,E1 22.514} C_DIS
LIN {X 0.087,Y -202.694,Z 448.103,A 0.000,B 0.000,C 90.000,E1 18.544} C_DIS
LIN {X 0.035,Y -198.366,Z 448.081,A 0.000,B 0.000,C 90.000,E1 14.537} C_DIS
LIN {X 0.012,Y -194.473,Z 448.054,A 0.000,B 0.000,C 90.000,E1 9.670} C_DIS
LIN {X -0.055,Y -191.619,Z 448.022,A 0.000,B 0.000,C 90.000,E1 3.955} C_DIS
LIN {X 0.073,Y -191.717,Z 447.965,A 0.000,B 0.000,C 90.000,E1 353.742} C_DIS
LIN {X 0.076,Y -194.659,Z 447.933,A 0.000,B 0.000,C 90.000,E1 347.993} C_DIS
LIN {X -0.066,Y -198.592,Z 447.906,A 0.000,B 0.000,C 90.000,E1 343.142} C_DIS
LIN {X -0.006,Y -202.868,Z 447.884,A 0.000,B 0.000,C 90.000,E1 339.082} C_DIS
LIN {X -0.086,Y -208.309,Z 447.862,A 0.000,B 0.000,C 90.000,E1 335.101} C_DIS
LIN {X -0.024,Y -214.479,Z 447.840,A 0.000,B 0.000,C 90.000,E1 331.129} C_DIS
LIN {X -0.104,Y -221.223,Z 447.818,A 0.000,B 0.000,C 90.000,E1 327.248} C_DIS
LIN {X 0.019,Y -228.679,Z 447.797,A 0.000,B 0.000,C 90.000,E1 323.371} C_DIS
LIN {X 0.021,Y -236.922,Z 447.776,A 0.000,B 0.000,C 90.000,E1 319.585} C_DIS
LIN {X -0.049,Y -244.201,Z 447.759,A 0.000,B 0.000,C 90.000,E1 316.620} C_DIS
LIN {X 0.058,Y -253.606,Z 447.741,A 0.000,B 0.000,C 90.000,E1 313.299} C_DIS
LIN {X -0.055,Y -264.228,Z 447.723,A 0.000,B 0.000,C 90.000,E1 310.092} C_DIS
LIN {X 0.002,Y -275.832,Z 447.705,A 0.000,B 0.000,C 90.000,E1 306.916} C_DIS
LIN {X -0.056,Y -288.331,Z 447.688,A 0.000,B 0.000,C 90.000,E1 303.833} C_DIS
LIN {X 0.021,Y -301.489,Z 447.671,A 0.000,B 0.000,C 90.000,E1 300.797} C_DIS
LIN {X 0.083,Y -317.257,Z 447.653,A 0.000,B 0.000,C 90.000,E1 297.513} C_DIS
LIN {X 0.076,Y -334.889,Z 447.635,A 0.000,B 0.000,C 90.000,E1 294.335} C_DIS
LIN {X 0.152,Y -346.451,Z 447.625,A 0.000,B 0.000,C 90.000,E1 292.461} C_DIS
LIN {X -0.036,Y -363.356,Z 447.611,A 0.000,B 0.000,C 90.000,E1 290.066} C_DIS
LIN {X 0.200,Y -386.572,Z 447.595,A 0.000,B 0.000,C 90.000,E1 287.094} C_DIS
LIN {X -0.136,Y -399.172,Z 447.587,A 0.000,B 0.000,C 90.000,E1 285.717} C_DIS
LIN {X -0.108,Y -424.864,Z 447.573,A 0.000,B 0.000,C 90.000,E1 283.119} C_DIS
LIN {X 0.192,Y -435.037,Z 447.567,A 0.000,B 0.000,C 90.000,E1 282.063} C_DIS
LIN {X -0.188,Y -444.845,Z 447.561,A 0.000,B 0.000,C 90.000,E1 281.074} C_DIS
LIN {X 0.066,Y -451.833,Z 447.557,A 0.000,B 0.000,C 90.000,E1 280.254} C_DIS
LIN {X -0.150,Y -458.353,Z 447.553,A 0.000,B 0.000,C 90.000,E1 279.500} C_DIS
LIN {X 0.153,Y -464.366,Z 447.548,A 0.000,B 0.000,C 90.000,E1 278.690} C_DIS
LIN {X 0.049,Y -469.823,Z 447.544,A 0.000,B 0.000,C 90.000,E1 277.936} C_DIS
LIN {X -0.005,Y -474.751,Z 447.540,A 0.000,B 0.000,C 90.000,E1 277.182} C_DIS
LIN {X -0.217,Y -480.593,Z 447.534,A 0.000,B 0.000,C 90.000,E1 276.201} C_DIS
LIN {X -0.194,Y -484.443,Z 447.530,A 0.000,B 0.000,C 90.000,E1 275.448} C_DIS
LIN {X -0.057,Y -486.701,Z 447.527,A 0.000,B 0.000,C 90.000,E1 274.935} C_DIS
LIN {X 0.140,Y -488.580,Z 447.525,A 0.000,B 0.000,C 90.000,E1 274.416} C_DIS
LIN {X -0.148,Y -490.111,Z 447.522,A 0.000,B 0.000,C 90.000,E1 273.955} C_DIS
LIN {X 0.030,Y -491.138,Z 447.519,A 0.000,B 0.000,C 90.000,E1 273.440} C_DIS
LIN {X 0.248,Y -491.784,Z 447.516,A 0.000,B 0.000,C 90.000,E1 272.922} C_DIS
LIN {X -0.046,Y -492.053,Z 447.514,A 0.000,B 0.000,C 90.000,E1 272.465} C_DIS
LIN {X 0.159,Y -491.931,Z 447.511,A 0.000,B 0.000,C 90.000,E1 271.949} C_DIS
LIN {X -0.111,Y -491.430,Z 447.508,A 0.000,B 0.000,C 90.000,E1 271.489} C_DIS
LIN {X 0.094,Y -490.518,Z 447.505,A 0.000,B 0.000,C 90.000,E1 270.974} C_DIS
LIN {X -0.192,Y -489.148,Z 447.503,A 0.000,B 0.000,C 90.000,E1 270.516} C_DIS
LIN {X 0.007,Y -487.259,Z 447.500,A 0.000,B 0.000,C 90.000,E1 270.000} C_DIS
LIN {X 0.196,Y -484.683,Z 447.497,A 0.000,B 0.000,C 90.000,E1 269.484} C_DIS
LIN {X -0.117,Y -481.403,Z 447.495,A 0.000,B 0.000,C 90.000,E1 269.026} C_DIS
LIN {X 0.035,Y -477.151,Z 447.492,A 0.000,B 0.000,C 90.000,E1 268.511} C_DIS
LIN {X 0.177,Y -471.844,Z 447.489,A 0.000,B 0.000,C 90.000,E1 267.993} C_DIS
LIN {X 0.165,Y -465.774,Z 447.486,A 0.000,B 0.000,C 90.000,E1 267.535} C_DIS
LIN {X 0.187,Y -459.103,Z 447.484,A 0.000,B 0.000,C 90.000,E1 267.135} C_DIS
LIN {X -0.142,Y -452.329,Z 447.482,A 0.000,B 0.000,C 90.000,E1 266.846} C_DIS
LIN {X -0.068,Y -445.318,Z 447.481,A 0.000,B 0.000,C 90.000,E1 266.560} C_DIS
LIN {X -0.100,Y -437.746,Z 447.480,A 0.000,B 0.000,C 90.000,E1 266.331} C_DIS
LIN {X -0.171,Y -429.400,Z 447.479,A 0.000,B 0.000,C 90.000,E1 266.159} C_DIS
LIN {X 0.178,Y -419.120,Z 447.478,A 0.000,B 0.000,C 90.000,E1 265.988} C_DIS
LIN {X 0.154,Y -408.947,Z 447.478,A 0.000,B 0.000,C 90.000,E1 265.931} C_DIS
LIN {X 0.111,Y -404.383,Z 447.477,A 0.000,B 0.000,C 90.000,E1 265.927} C_DIS
LIN {X 0.018,Y -180.918,Z 447.477,A 0.000,B 0.000,C 90.000,E1 265.927} C_DIS
LIN {X 0.051,Y -180.839,Z 447.472,A 0.000,B 0.000,C 90.000,E1 264.894} C_DIS
LIN {X -0.052,Y -178.880,Z 447.443,A 0.000,B 0.000,C 90.000,E1 259.690} C_DIS
LIN {X 0.024,Y -175.922,Z 447.414,A 0.000,B 0.000,C 90.000,E1 254.574} C_DIS
LIN {X -0.087,Y -174.621,Z 447.405,A 0.000,B 0.000,C 90.000,E1 252.906} C_DIS
LIN {X 0.005,Y -171.601,Z 447.381,A 0.000,B 0.000,C 90.000,E1 248.592} C_DIS
LIN {X -0.006,Y -167.824,Z 447.357,A 0.000,B 0.000,C 90.000,E1 244.280} C_DIS
LIN {X 0.011,Y -166.548,Z 447.347,A 0.000,B 0.000,C 90.000,E1 242.538} C_DIS
LIN {X -0.078,Y -162.544,Z 447.323,A 0.000,B 0.000,C 90.000,E1 238.201} C_DIS
LIN {X -0.018,Y -161.222,Z 447.313,A 0.000,B 0.000,C 90.000,E1 236.421} C_DIS
LIN {X 0.017,Y -157.229,Z 447.289,A 0.000,B 0.000,C 90.000,E1 231.984} C_DIS
LIN {X 0.041,Y -155.954,Z 447.279,A 0.000,B 0.000,C 90.000,E1 230.194} C_DIS
LIN {X -0.001,Y -152.206,Z 447.254,A 0.000,B 0.000,C 90.000,E1 225.729} C_DIS
LIN {X 0.020,Y -150.452,Z 447.239,A 0.000,B 0.000,C 90.000,E1 223.014} C_DIS
LIN {X 0.046,Y -147.178,Z 447.214,A 0.000,B 0.000,C 90.000,E1 218.463} C_DIS
LIN {X 0.014,Y -145.195,Z 447.193,A 0.000,B 0.000,C 90.000,E1 214.818} C_DIS
LIN {X 0.048,Y -142.335,Z 447.163,A 0.000,B 0.000,C 90.000,E1 209.283} C_DIS
LIN {X -0.023,Y -141.723,Z 447.153,A 0.000,B 0.000,C 90.000,E1 207.462} C_DIS
LIN {X -0.041,Y -139.478,Z 447.116,A 0.000,B 0.000,C 90.000,E1 200.972} C_DIS
LIN {X -0.052,Y -138.976,Z 447.101,A 0.000,B 0.000,C 90.000,E1 198.181} C_DIS
LIN {X 0.070,Y -138.331,Z 447.054,A 0.000,B 0.000,C 90.000,E1 189.726} C_DIS
LIN {X -0.066,Y -139.432,Z 447.007,A 0.000,B 0.000,C 90.000,E1 181.375} C_DIS
LIN {X 0.014,Y -140.958,Z 446.976,A 0.000,B 0.000,C 90.000,E1 175.755} C_DIS
LIN {X -0.036,Y -142.714,Z 446.956,A 0.000,B 0.000,C 90.000,E1 172.064} C_DIS
LIN {X 0.063,Y -145.091,Z 446.930,A 0.000,B 0.000,C 90.000,E1 167.409} C_DIS
LIN {X 0.059,Y -147.715,Z 446.910,A 0.000,B 0.000,C 90.000,E1 163.740} C_DIS
LIN {X 0.000,Y -150.373,Z 446.890,A 0.000,B 0.000,C 90.000,E1 160.115} C_DIS
LIN {X 0.018,Y -153.801,Z 446.869,A 0.000,B 0.000,C 90.000,E1 156.485} C_DIS
LIN {X 0.077,Y -157.213,Z 446.849,A 0.000,B 0.000,C 90.000,E1 152.871} C_DIS
LIN {X 0.019,Y -161.377,Z 446.830,A 0.000,B 0.000,C 90.000,E1 149.331} C_DIS
LIN {X 0.030,Y -165.579,Z 446.810,A 0.000,B 0.000,C 90.000,E1 145.801} C_DIS
LIN {X 0.017,Y -170.500,Z 446.791,A 0.000,B 0.000,C 90.000,E1 142.316} C_DIS
LIN {X 0.061,Y -175.380,Z 446.772,A 0.000,B 0.000,C 90.000,E1 138.852} C_DIS
LIN {X -0.077,Y -181.004,Z 446.753,A 0.000,B 0.000,C 90.000,E1 135.486} C_DIS
LIN {X 0.048,Y -186.433,Z 446.734,A 0.000,B 0.000,C 90.000,E1 132.081} C_DIS
LIN {X 0.117,Y -191.059,Z 446.720,A 0.000,B 0.000,C 90.000,E1 129.564} C_DIS
LIN {X 0.028,Y -195.240,Z 446.706,A 0.000,B 0.000,C 90.000,E1 127.156} C_DIS
LIN {X 0.010,Y -292.872,Z 446.706,A 0.000,B 0.000,C 90.000,E1 127.156} C_DIS
LIN {X -0.151,Y -295.075,Z 446.706,A 0.000,B 0.000,C 90.000,E1 127.156} C_DIS
LIN {X 0.014,Y -298.247,Z 446.706,A 0.000,B 0.000,C 90.000,E1 126.996} C_DIS
LIN {X 0.005,Y -301.616,Z 446.704,A 0.000,B 0.000,C 90.000,E1 126.744} C_DIS
LIN {X -0.004,Y -305.291,Z 446.702,A 0.000,B 0.000,C 90.000,E1 126.297} C_DIS
LIN {X 0.023,Y -307.178,Z 446.700,A 0.000,B 0.000,C 90.000,E1 125.964} C_DIS
LIN {X -0.020,Y -308.657,Z 446.698,A 0.000,B 0.000,C 90.000,E1 125.644} C_DIS
LIN {X 0.051,Y -310.819,Z 446.694,A 0.000,B 0.000,C 90.000,E1 124.978} C_DIS
LIN {X 0.047,Y -321.545,Z 446.676,A 0.000,B 0.000,C 90.000,E1 121.750} C_DIS
LIN {X 0.050,Y -332.571,Z 446.661,A 0.000,B 0.000,C 90.000,E1 118.899} C_DIS
LIN {X 0.040,Y -345.007,Z 446.645,A 0.000,B 0.000,C 90.000,E1 116.104} C_DIS
LIN {X -0.126,Y -357.333,Z 446.632,A 0.000,B 0.000,C 90.000,E1 113.695} C_DIS
LIN {X 0.056,Y -370.950,Z 446.618,A 0.000,B 0.000,C 90.000,E1 111.280} C_DIS
LIN {X -0.028,Y -385.955,Z 446.605,A 0.000,B 0.000,C 90.000,E1 108.960} C_DIS
LIN {X 0.012,Y -402.459,Z 446.593,A 0.000,B 0.000,C 90.000,E1 106.677} C_DIS
LIN {X -0.154,Y -420.586,Z 446.580,A 0.000,B 0.000,C 90.000,E1 104.481} C_DIS
LIN {X 0.172,Y -440.280,Z 446.568,A 0.000,B 0.000,C 90.000,E1 102.299} C_DIS
LIN {X -0.131,Y -460.676,Z 446.557,A 0.000,B 0.000,C 90.000,E1 100.366} C_DIS
LIN {X -0.109,Y -484.162,Z 446.546,A 0.000,B 0.000,C 90.000,E1 98.341} C_DIS
LIN {X 0.068,Y -486.204,Z 446.545,A 0.000,B 0.000,C 90.000,E1 98.106} C_DIS
LIN {X -0.046,Y -487.990,Z 446.544,A 0.000,B 0.000,C 90.000,E1 97.871} C_DIS
LIN {X -0.227,Y -489.330,Z 446.542,A 0.000,B 0.000,C 90.000,E1 97.644} C_DIS
LIN {X -0.016,Y -491.001,Z 446.540,A 0.000,B 0.000,C 90.000,E1 97.125} C_DIS
LIN {X 0.205,Y -491.588,Z 446.537,A 0.000,B 0.000,C 90.000,E1 96.606} C_DIS
LIN {X -0.052,Y -491.191,Z 446.534,A 0.000,B 0.000,C 90.000,E1 96.144} C_DIS
LIN {X 0.181,Y -489.745,Z 446.531,A 0.000,B 0.000,C 90.000,E1 95.625} C_DIS
LIN {X 0.075,Y -488.553,Z 446.530,A 0.000,B 0.000,C 90.000,E1 95.391} C_DIS
LIN {X -0.077,Y -486.959,Z 446.529,A 0.000,B 0.000,C 90.000,E1 95.163} C_DIS
LIN {X 0.143,Y -477.066,Z 446.522,A 0.000,B 0.000,C 90.000,E1 93.898} C_DIS
LIN {X 0.097,Y -457.465,Z 446.508,A 0.000,B 0.000,C 90.000,E1 91.375} C_DIS
LIN {X -0.170,Y -445.121,Z 446.498,A 0.000,B 0.000,C 90.000,E1 89.599} C_DIS
LIN {X 0.209,Y -433.522,Z 446.487,A 0.000,B 0.000,C 90.000,E1 87.707} C_DIS
LIN {X -0.113,Y -417.300,Z 446.473,A 0.000,B 0.000,C 90.000,E1 85.065} C_DIS
LIN {X -0.091,Y -403.395,Z 446.459,A 0.000,B 0.000,C 90.000,E1 82.591} C_DIS
LIN {X -0.024,Y -392.666,Z 446.448,A 0.000,B 0.000,C 90.000,E1 80.622} C_DIS
LIN {X -0.007,Y -380.466,Z 446.435,A 0.000,B 0.000,C 90.000,E1 78.342} C_DIS
LIN {X 0.145,Y -365.721,Z 446.419,A 0.000,B 0.000,C 90.000,E1 75.408} C_DIS
LIN {X -0.116,Y -352.079,Z 446.403,A 0.000,B 0.000,C 90.000,E1 72.472} C_DIS
LIN {X 0.116,Y -337.243,Z 446.382,A 0.000,B 0.000,C 90.000,E1 68.773} C_DIS
LIN {X 0.019,Y -329.008,Z 446.370,A 0.000,B 0.000,C 90.000,E1 66.613} C_DIS
LIN {X 0.087,Y -319.728,Z 446.356,A 0.000,B 0.000,C 90.000,E1 64.076} C_DIS
LIN {X 0.066,Y -310.728,Z 446.342,A 0.000,B 0.000,C 90.000,E1 61.513} C_DIS
LIN {X 0.001,Y -301.895,Z 446.327,A 0.000,B 0.000,C 90.000,E1 58.918} C_DIS
LIN {X 0.062,Y -291.545,Z 446.309,A 0.000,B 0.000,C 90.000,E1 55.595} C_DIS
LIN {X -0.175,Y -281.988,Z 446.290,A 0.000,B 0.000,C 90.000,E1 52.271} C_DIS
LIN {X -0.054,Y -276.234,Z 446.279,A 0.000,B 0.000,C 90.000,E1 50.194} C_DIS
LIN {X 0.132,Y -270.291,Z 446.267,A 0.000,B 0.000,C 90.000,E1 48.081} C_DIS
LIN {X 0.179,Y -264.127,Z 446.256,A 0.000,B 0.000,C 90.000,E1 45.972} C_DIS
LIN {X 0.102,Y -257.788,Z 446.244,A 0.000,B 0.000,C 90.000,E1 43.866} C_DIS
LIN {X -0.078,Y -251.319,Z 446.232,A 0.000,B 0.000,C 90.000,E1 41.757} C_DIS
LIN {X 0.006,Y -242.758,Z 446.216,A 0.000,B 0.000,C 90.000,E1 38.830} C_DIS
LIN {X -0.045,Y -234.555,Z 446.199,A 0.000,B 0.000,C 90.000,E1 35.884} C_DIS
LIN {X -0.056,Y -227.080,Z 446.183,A 0.000,B 0.000,C 90.000,E1 32.880} C_DIS
LIN {X 0.067,Y -220.458,Z 446.166,A 0.000,B 0.000,C 90.000,E1 29.795} C_DIS
LIN {X -0.105,Y -214.600,Z 446.148,A 0.000,B 0.000,C 90.000,E1 26.744} C_DIS
LIN {X 0.087,Y -208.283,Z 446.127,A 0.000,B 0.000,C 90.000,E1 22.770} C_DIS
LIN {X -0.050,Y -202.983,Z 446.105,A 0.000,B 0.000,C 90.000,E1 18.833} C_DIS
LIN {X 0.093,Y -198.571,Z 446.082,A 0.000,B 0.000,C 90.000,E1 14.773} C_DIS
LIN {X 0.078,Y -194.569,Z 446.055,A 0.000,B 0.000,C 90.000,E1 9.905} C_DIS
LIN {X 0.024,Y -191.614,Z 446.023,A 0.000,B 0.000,C 90.000,E1 4.188} C_DIS
LIN {X 0.067,Y -191.597,Z 445.965,A 0.000,B 0.000,C 90.000,E1 353.742} C_DIS
LIN {X 0.066,Y -194.524,Z 445.933,A 0.000,B 0.000,C 90.000,E1 347.993} C_DIS
LIN {X -0.081,Y -198.441,Z 445.906,A 0.000,B 0.000,C 90.000,E1 343.142} C_DIS
LIN {X -0.027,Y -202.697,Z 445.884,A 0.000,B 0.000,C 90.000,E1 339.082} C_DIS
LIN {X 0.076,Y -208.154,Z 445.862,A 0.000,B 0.000,C 90.000,E1 335.049} C_DIS
LIN {X -0.056,Y -214.332,Z 445.840,A 0.000,B 0.000,C 90.000,E1 331.129} C_DIS
LIN {X 0.045,Y -221.073,Z 445.818,A 0.000,B 0.000,C 90.000,E1 327.199} C_DIS
LIN {X 0.112,Y -228.528,Z 445.796,A 0.000,B 0.000,C 90.000,E1 323.336} C_DIS
LIN {X -0.029,Y -236.792,Z 445.775,A 0.000,B 0.000,C 90.000,E1 319.585} C_DIS
LIN {X -0.105,Y -244.080,Z 445.759,A 0.000,B 0.000,C 90.000,E1 316.620} C_DIS
LIN {X -0.003,Y -253.499,Z 445.741,A 0.000,B 0.000,C 90.000,E1 313.299} C_DIS
LIN {X -0.121,Y -264.137,Z 445.723,A 0.000,B 0.000,C 90.000,E1 310.092} C_DIS
LIN {X 0.151,Y -275.764,Z 445.705,A 0.000,B 0.000,C 90.000,E1 306.870} C_DIS
LIN {X 0.108,Y -288.284,Z 445.688,A 0.000,B 0.000,C 90.000,E1 303.785} C_DIS
LIN {X -0.061,Y -301.465,Z 445.671,A 0.000,B 0.000,C 90.000,E1 300.797} C_DIS
LIN {X -0.003,Y -317.258,Z 445.653,A 0.000,B 0.000,C 90.000,E1 297.513} C_DIS
LIN {X -0.013,Y -334.888,Z 445.635,A 0.000,B 0.000,C 90.000,E1 294.335} C_DIS
LIN {X 0.060,Y -346.490,Z 445.625,A 0.000,B 0.000,C 90.000,E1 292.461} C_DIS
LIN {X -0.065,Y -361.194,Z 445.613,A 0.000,B 0.000,C 90.000,E1 290.355} C_DIS
LIN {X -0.030,Y -384.247,Z 445.597,A 0.000,B 0.000,C 90.000,E1 287.402} C_DIS
LIN {X 0.139,Y -396.445,Z 445.589,A 0.000,B 0.000,C 90.000,E1 285.969} C_DIS
LIN {X 0.028,Y -422.253,Z 445.574,A 0.000,B 0.000,C 90.000,E1 283.355} C_DIS
LIN {X 0.036,Y -432.432,Z 445.569,A 0.000,B 0.000,C 90.000,E1 282.355} C_DIS
LIN {X -0.008,Y -439.875,Z 445.564,A 0.000,B 0.000,C 90.000,E1 281.591} C_DIS
LIN {X -0.064,Y -449.489,Z 445.559,A 0.000,B 0.000,C 90.000,E1 280.546} C_DIS
LIN {X 0.232,Y -456.149,Z 445.554,A 0.000,B 0.000,C 90.000,E1 279.726} C_DIS
LIN {X 0.053,Y -462.322,Z 445.550,A 0.000,B 0.000,C 90.000,E1 278.973} C_DIS
LIN {X -0.069,Y -467.984,Z 445.546,A 0.000,B 0.000,C 90.000,E1 278.219} C_DIS
LIN {X -0.149,Y -473.075,Z 445.541,A 0.000,B 0.000,C 90.000,E1 277.466} C_DIS
LIN {X 0.089,Y -479.169,Z 445.536,A 0.000,B 0.000,C 90.000,E1 276.429} C_DIS
LIN {X 0.058,Y -483.194,Z 445.532,A 0.000,B 0.000,C 90.000,E1 275.682} C_DIS
LIN {X 0.060,Y -486.684,Z 445.527,A 0.000,B 0.000,C 90.000,E1 274.935} C_DIS
LIN {X -0.230,Y -488.604,Z 445.525,A 0.000,B 0.000,C 90.000,E1 274.473} C_DIS
LIN {X -0.031,Y -490.081,Z 445.522,A 0.000,B 0.000,C 90.000,E1 273.955} C_DIS
LIN {X 0.149,Y -491.109,Z 445.519,A 0.000,B 0.000,C 90.000,E1 273.440} C_DIS
LIN {X -0.124,Y -491.775,Z 445.516,A 0.000,B 0.000,C 90.000,E1 272.980} C_DIS
LIN {X 0.073,Y -492.042,Z 445.514,A 0.000,B 0.000,C 90.000,E1 272.465} C_DIS
LIN {X -0.214,Y -491.934,Z 445.511,A 0.000,B 0.000,C 90.000,E1 272.007} C_DIS
LIN {X 0.007,Y -491.445,Z 445.508,A 0.000,B 0.000,C 90.000,E1 271.489} C_DIS
LIN {X 0.213,Y -490.561,Z 445.506,A 0.000,B 0.000,C 90.000,E1 270.974} C_DIS
LIN {X -0.074,Y -489.222,Z 445.503,A 0.000,B 0.000,C 90.000,E1 270.516} C_DIS
LIN {X 0.124,Y -487.331,Z 445.500,A 0.000,B 0.000,C 90.000,E1 270.000} C_DIS
LIN {X -0.024,Y -486.203,Z 445.499,A 0.000,B 0.000,C 90.000,E1 269.771} C_DIS
LIN {X 0.156,Y -483.276,Z 445.496,A 0.000,B 0.000,C 90.000,E1 269.255} C_DIS
LIN {X 0.000,Y -481.578,Z 445.495,A 0.000,B 0.000,C 90.000,E1 269.026} C_DIS
LIN {X 0.152,Y -477.390,Z 445.492,A 0.000,B 0.000,C 90.000,E1 268.511} C_DIS
LIN {X -0.022,Y -474.927,Z 445.490,A 0.000,B 0.000,C 90.000,E1 268.282} C_DIS
LIN {X -0.189,Y -469.279,Z 445.488,A 0.000,B 0.000,C 90.000,E1 267.822} C_DIS
LIN {X -0.199,Y -466.091,Z 445.486,A 0.000,B 0.000,C 90.000,E1 267.593} C_DIS
LIN {X -0.178,Y -459.470,Z 445.484,A 0.000,B 0.000,C 90.000,E1 267.192} C_DIS
LIN {X -0.066,Y -452.636,Z 445.482,A 0.000,B 0.000,C 90.000,E1 266.846} C_DIS
LIN {X -0.001,Y -445.564,Z 445.481,A 0.000,B 0.000,C 90.000,E1 266.560} C_DIS
LIN {X -0.011,Y -438.223,Z 445.480,A 0.000,B 0.000,C 90.000,E1 266.331} C_DIS
LIN {X -0.091,Y -430.001,Z 445.479,A 0.000,B 0.000,C 90.000,E1 266.159} C_DIS
LIN {X -0.190,Y -419.860,Z 445.478,A 0.000,B 0.000,C 90.000,E1 266.045} C_DIS
LIN {X 0.146,Y -406.979,Z 445.477,A 0.000,B 0.000,C 90.000,E1 265.927} C_DIS
LIN {X 0.032,Y -180.918,Z 445.477,A 0.000,B 0.000,C 90.000,E1 265.927} C_DIS
LIN {X 0.064,Y -180.840,Z 445.472,A 0.000,B 0.000,C 90.000,E1 264.894} C_DIS
LIN {X -0.040,Y -178.881,Z 445.443,A 0.000,B 0.000,C 90.000,E1 259.690} C_DIS
LIN {X 0.037,Y -175.924,Z 445.414,A 0.000,B 0.000,C 90.000,E1 254.574} C_DIS
LIN {X -0.018,Y -175.363,Z 445.410,A 0.000,B 0.000,C 90.000,E1 253.740} C_DIS
LIN {X 0.040,Y -172.141,Z 445.386,A 0.000,B 0.000,C 90.000,E1 249.444} C_DIS
LIN {X 0.018,Y -171.605,Z 445.381,A 0.000,B 0.000,C 90.000,E1 248.592} C_DIS
LIN {X 0.006,Y -167.827,Z 445.357,A 0.000,B 0.000,C 90.000,E1 244.280} C_DIS
LIN {X 0.024,Y -166.553,Z 445.347,A 0.000,B 0.000,C 90.000,E1 242.538} C_DIS
LIN {X -0.066,Y -162.548,Z 445.323,A 0.000,B 0.000,C 90.000,E1 238.201} C_DIS
LIN {X -0.006,Y -161.226,Z 445.313,A 0.000,B 0.000,C 90.000,E1 236.421} C_DIS
LIN {X 0.030,Y -157.232,Z 445.289,A 0.000,B 0.000,C 90.000,E1 231.984} C_DIS
LIN {X 0.052,Y -155.957,Z 445.279,A 0.000,B 0.000,C 90.000,E1 230.194} C_DIS
LIN {X 0.011,Y -152.210,Z 445.254,A 0.000,B 0.000,C 90.000,E1 225.729} C_DIS
LIN {X 0.032,Y -150.455,Z 445.239,A 0.000,B 0.000,C 90.000,E1 223.014} C_DIS
LIN {X 0.058,Y -147.181,Z 445.214,A 0.000,B 0.000,C 90.000,E1 218.463} C_DIS
LIN {X 0.025,Y -145.198,Z 445.193,A 0.000,B 0.000,C 90.000,E1 214.818} C_DIS
LIN {X 0.059,Y -142.336,Z 445.163,A 0.000,B 0.000,C 90.000,E1 209.283} C_DIS
LIN {X -0.012,Y -141.725,Z 445.153,A 0.000,B 0.000,C 90.000,E1 207.462} C_DIS
LIN {X -0.029,Y -139.479,Z 445.116,A 0.000,B 0.000,C 90.000,E1 200.972} C_DIS
LIN {X -0.041,Y -138.978,Z 445.101,A 0.000,B 0.000,C 90.000,E1 198.181} C_DIS
LIN {X -0.055,Y -138.332,Z 445.054,A 0.000,B 0.000,C 90.000,E1 189.782} C_DIS
LIN {X -0.055,Y -139.431,Z 445.008,A 0.000,B 0.000,C 90.000,E1 181.375} C_DIS
LIN {X -0.002,Y -141.359,Z 444.971,A 0.000,B 0.000,C 90.000,E1 174.837} C_DIS
LIN {X -0.026,Y -142.712,Z 444.956,A 0.000,B 0.000,C 90.000,E1 172.064} C_DIS
LIN {X -0.067,Y -145.088,Z 444.930,A 0.000,B 0.000,C 90.000,E1 167.465} C_DIS
LIN {X 0.070,Y -147.713,Z 444.910,A 0.000,B 0.000,C 90.000,E1 163.740} C_DIS
LIN {X 0.011,Y -150.369,Z 444.890,A 0.000,B 0.000,C 90.000,E1 160.115} C_DIS
LIN {X 0.029,Y -153.796,Z 444.869,A 0.000,B 0.000,C 90.000,E1 156.485} C_DIS
LIN {X -0.051,Y -157.208,Z 444.849,A 0.000,B 0.000,C 90.000,E1 152.922} C_DIS
LIN {X 0.031,Y -161.371,Z 444.830,A 0.000,B 0.000,C 90.000,E1 149.331} C_DIS
LIN {X 0.042,Y -165.574,Z 444.810,A 0.000,B 0.000,C 90.000,E1 145.801} C_DIS
LIN {X 0.029,Y -170.493,Z 444.791,A 0.000,B 0.000,C 90.000,E1 142.316} C_DIS
LIN {X 0.075,Y -175.373,Z 444.772,A 0.000,B 0.000,C 90.000,E1 138.852} C_DIS
LIN {X -0.063,Y -180.998,Z 444.753,A 0.000,B 0.000,C 90.000,E1 135.486} C_DIS
LIN {X 0.061,Y -186.426,Z 444.734,A 0.000,B 0.000,C 90.000,E1 132.081} C_DIS
LIN {X 0.009,Y -191.052,Z 444.720,A 0.000,B 0.000,C 90.000,E1 129.600} C_DIS
LIN {X 0.093,Y -195.352,Z 444.706,A 0.000,B 0.000,C 90.000,E1 127.076} C_DIS
LIN {X 0.086,Y -294.024,Z 444.706,A 0.000,B 0.000,C 90.000,E1 127.076} C_DIS
LIN {X -0.078,Y -295.562,Z 444.706,A 0.000,B 0.000,C 90.000,E1 127.076} C_DIS
LIN {X 0.021,Y -299.479,Z 444.705,A 0.000,B 0.000,C 90.000,E1 126.870} C_DIS
LIN {X 0.122,Y -301.776,Z 444.704,A 0.000,B 0.000,C 90.000,E1 126.664} C_DIS
LIN {X 0.082,Y -304.948,Z 444.702,A 0.000,B 0.000,C 90.000,E1 126.297} C_DIS
LIN {X -0.098,Y -306.908,Z 444.700,A 0.000,B 0.000,C 90.000,E1 126.011} C_DIS
LIN {X -0.030,Y -308.443,Z 444.698,A 0.000,B 0.000,C 90.000,E1 125.678} C_DIS
LIN {X -0.034,Y -310.703,Z 444.695,A 0.000,B 0.000,C 90.000,E1 125.025} C_DIS
LIN {X -0.055,Y -321.413,Z 444.677,A 0.000,B 0.000,C 90.000,E1 121.799} C_DIS
LIN {X -0.068,Y -332.425,Z 444.661,A 0.000,B 0.000,C 90.000,E1 118.949} C_DIS
LIN {X -0.093,Y -344.846,Z 444.645,A 0.000,B 0.000,C 90.000,E1 116.155} C_DIS
LIN {X 0.052,Y -357.157,Z 444.632,A 0.000,B 0.000,C 90.000,E1 113.695} C_DIS
LIN {X -0.109,Y -370.757,Z 444.618,A 0.000,B 0.000,C 90.000,E1 111.334} C_DIS
LIN {X 0.155,Y -385.745,Z 444.605,A 0.000,B 0.000,C 90.000,E1 108.960} C_DIS
LIN {X 0.197,Y -402.231,Z 444.593,A 0.000,B 0.000,C 90.000,E1 106.677} C_DIS
LIN {X 0.034,Y -420.337,Z 444.580,A 0.000,B 0.000,C 90.000,E1 104.481} C_DIS
LIN {X -0.075,Y -440.017,Z 444.569,A 0.000,B 0.000,C 90.000,E1 102.355} C_DIS
LIN {X 0.045,Y -460.406,Z 444.558,A 0.000,B 0.000,C 90.000,E1 100.366} C_DIS
LIN {X 0.057,Y -483.925,Z 444.546,A 0.000,B 0.000,C 90.000,E1 98.341} C_DIS
LIN {X 0.233,Y -486.066,Z 444.545,A 0.000,B 0.000,C 90.000,E1 98.106} C_DIS
LIN {X 0.152,Y -487.900,Z 444.544,A 0.000,B 0.000,C 90.000,E1 97.871} C_DIS
LIN {X 0.005,Y -489.282,Z 444.542,A 0.000,B 0.000,C 90.000,E1 97.644} C_DIS
LIN {X 0.216,Y -491.058,Z 444.540,A 0.000,B 0.000,C 90.000,E1 97.125} C_DIS
LIN {X -0.051,Y -491.733,Z 444.537,A 0.000,B 0.000,C 90.000,E1 96.663} C_DIS
LIN {X 0.180,Y -491.422,Z 444.534,A 0.000,B 0.000,C 90.000,E1 96.144} C_DIS
LIN {X -0.074,Y -490.075,Z 444.532,A 0.000,B 0.000,C 90.000,E1 95.682} C_DIS
LIN {X -0.178,Y -488.943,Z 444.530,A 0.000,B 0.000,C 90.000,E1 95.448} C_DIS
LIN {X 0.156,Y -487.425,Z 444.529,A 0.000,B 0.000,C 90.000,E1 95.163} C_DIS
LIN {X 0.040,Y -479.593,Z 444.523,A 0.000,B 0.000,C 90.000,E1 94.188} C_DIS
LIN {X -0.172,Y -461.747,Z 444.511,A 0.000,B 0.000,C 90.000,E1 91.949} C_DIS
LIN {X 0.109,Y -448.940,Z 444.501,A 0.000,B 0.000,C 90.000,E1 90.115} C_DIS
LIN {X 0.022,Y -433.913,Z 444.488,A 0.000,B 0.000,C 90.000,E1 87.764} C_DIS
LIN {X -0.181,Y -416.130,Z 444.471,A 0.000,B 0.000,C 90.000,E1 84.837} C_DIS
LIN {X 0.159,Y -403.781,Z 444.459,A 0.000,B 0.000,C 90.000,E1 82.591} C_DIS
LIN {X -0.161,Y -393.071,Z 444.448,A 0.000,B 0.000,C 90.000,E1 80.679} C_DIS
LIN {X -0.129,Y -380.884,Z 444.435,A 0.000,B 0.000,C 90.000,E1 78.398} C_DIS
LIN {X 0.062,Y -367.582,Z 444.421,A 0.000,B 0.000,C 90.000,E1 75.755} C_DIS
LIN {X 0.101,Y -353.790,Z 444.404,A 0.000,B 0.000,C 90.000,E1 72.779} C_DIS
LIN {X 0.055,Y -339.955,Z 444.386,A 0.000,B 0.000,C 90.000,E1 69.444} C_DIS
LIN {X 0.000,Y -330.468,Z 444.372,A 0.000,B 0.000,C 90.000,E1 66.975} C_DIS
LIN {X -0.027,Y -321.124,Z 444.358,A 0.000,B 0.000,C 90.000,E1 64.460} C_DIS
LIN {X -0.009,Y -312.049,Z 444.344,A 0.000,B 0.000,C 90.000,E1 61.897} C_DIS
LIN {X 0.068,Y -303.156,Z 444.329,A 0.000,B 0.000,C 90.000,E1 59.282} C_DIS
LIN {X -0.091,Y -291.695,Z 444.309,A 0.000,B 0.000,C 90.000,E1 55.674} C_DIS
LIN {X 0.074,Y -282.130,Z 444.290,A 0.000,B 0.000,C 90.000,E1 52.271} C_DIS
LIN {X 0.015,Y -276.390,Z 444.279,A 0.000,B 0.000,C 90.000,E1 50.231} C_DIS
LIN {X -0.006,Y -270.461,Z 444.268,A 0.000,B 0.000,C 90.000,E1 48.162} C_DIS
LIN {X 0.046,Y -264.299,Z 444.256,A 0.000,B 0.000,C 90.000,E1 46.053} C_DIS
LIN {X -0.023,Y -257.975,Z 444.244,A 0.000,B 0.000,C 90.000,E1 43.947} C_DIS
LIN {X 0.159,Y -251.521,Z 444.232,A 0.000,B 0.000,C 90.000,E1 41.757} C_DIS
LIN {X -0.103,Y -242.954,Z 444.216,A 0.000,B 0.000,C 90.000,E1 38.910} C_DIS
LIN {X -0.010,Y -232.791,Z 444.195,A 0.000,B 0.000,C 90.000,E1 35.185} C_DIS
LIN {X 0.123,Y -225.519,Z 444.179,A 0.000,B 0.000,C 90.000,E1 32.133} C_DIS
LIN {X 0.091,Y -219.087,Z 444.162,A 0.000,B 0.000,C 90.000,E1 29.077} C_DIS
LIN {X 0.076,Y -213.386,Z 444.144,A 0.000,B 0.000,C 90.000,E1 25.976} C_DIS
LIN {X -0.052,Y -207.246,Z 444.123,A 0.000,B 0.000,C 90.000,E1 22.078} C_DIS
LIN {X 0.091,Y -202.079,Z 444.100,A 0.000,B 0.000,C 90.000,E1 18.055} C_DIS
LIN {X -0.038,Y -197.844,Z 444.078,A 0.000,B 0.000,C 90.000,E1 14.064} C_DIS
LIN {X 0.076,Y -193.991,Z 444.051,A 0.000,B 0.000,C 90.000,E1 9.151} C_DIS
LIN {X -0.083,Y -191.035,Z 444.014,A 0.000,B 0.000,C 90.000,E1 2.636} C_DIS
LIN {X 0.019,Y -191.788,Z 443.961,A 0.000,B 0.000,C 90.000,E1 352.932} C_DIS
LIN {X 0.061,Y -194.959,Z 443.929,A 0.000,B 0.000,C 90.000,E1 347.173} C_DIS
LIN {X -0.096,Y -198.295,Z 443.906,A 0.000,B 0.000,C 90.000,E1 343.142} C_DIS
LIN {X -0.047,Y -202.563,Z 443.884,A 0.000,B 0.000,C 90.000,E1 339.082} C_DIS
LIN {X 0.050,Y -208.002,Z 443.861,A 0.000,B 0.000,C 90.000,E1 335.049} C_DIS
LIN {X -0.088,Y -214.187,Z 443.839,A 0.000,B 0.000,C 90.000,E1 331.129} C_DIS
LIN {X 0.008,Y -220.934,Z 443.818,A 0.000,B 0.000,C 90.000,E1 327.199} C_DIS
LIN {X 0.068,Y -228.376,Z 443.796,A 0.000,B 0.000,C 90.000,E1 323.336} C_DIS
LIN {X 0.102,Y -236.659,Z 443.775,A 0.000,B 0.000,C 90.000,E1 319.542} C_DIS
LIN {X -0.008,Y -244.951,Z 443.757,A 0.000,B 0.000,C 90.000,E1 316.215} C_DIS
LIN {X -0.044,Y -254.524,Z 443.738,A 0.000,B 0.000,C 90.000,E1 312.933} C_DIS
LIN {X -0.124,Y -265.297,Z 443.721,A 0.000,B 0.000,C 90.000,E1 309.725} C_DIS
LIN {X 0.014,Y -277.060,Z 443.703,A 0.000,B 0.000,C 90.000,E1 306.537} C_DIS
LIN {X 0.014,Y -289.672,Z 443.686,A 0.000,B 0.000,C 90.000,E1 303.452} C_DIS
LIN {X -0.122,Y -302.957,Z 443.669,A 0.000,B 0.000,C 90.000,E1 300.463} C_DIS
LIN {X -0.022,Y -318.936,Z 443.651,A 0.000,B 0.000,C 90.000,E1 297.180} C_DIS
LIN {X 0.013,Y -336.744,Z 443.633,A 0.000,B 0.000,C 90.000,E1 294.003} C_DIS
LIN {X -0.018,Y -348.573,Z 443.623,A 0.000,B 0.000,C 90.000,E1 292.153} C_DIS
LIN {X -0.095,Y -363.472,Z 443.611,A 0.000,B 0.000,C 90.000,E1 290.047} C_DIS
LIN {X -0.122,Y -384.326,Z 443.597,A 0.000,B 0.000,C 90.000,E1 287.402} C_DIS
LIN {X -0.021,Y -396.620,Z 443.589,A 0.000,B 0.000,C 90.000,E1 285.969} C_DIS
LIN {X -0.052,Y -424.835,Z 443.573,A 0.000,B 0.000,C 90.000,E1 283.119} C_DIS
LIN {X 0.042,Y -432.492,Z 443.569,A 0.000,B 0.000,C 90.000,E1 282.355} C_DIS
LIN {X 0.012,Y -439.905,Z 443.564,A 0.000,B 0.000,C 90.000,E1 281.591} C_DIS
LIN {X -0.055,Y -449.541,Z 443.559,A 0.000,B 0.000,C 90.000,E1 280.546} C_DIS
LIN {X 0.240,Y -456.181,Z 443.554,A 0.000,B 0.000,C 90.000,E1 279.726} C_DIS
LIN {X 0.062,Y -462.335,Z 443.550,A 0.000,B 0.000,C 90.000,E1 278.973} C_DIS
LIN {X -0.060,Y -467.988,Z 443.546,A 0.000,B 0.000,C 90.000,E1 278.219} C_DIS
LIN {X -0.141,Y -473.080,Z 443.541,A 0.000,B 0.000,C 90.000,E1 277.466} C_DIS
LIN {X 0.098,Y -479.188,Z 443.536,A 0.000,B 0.000,C 90.000,E1 276.429} C_DIS
LIN {X 0.067,Y -483.225,Z 443.532,A 0.000,B 0.000,C 90.000,E1 275.682} C_DIS
LIN {X 0.069,Y -486.703,Z 443.527,A 0.000,B 0.000,C 90.000,E1 274.935} C_DIS
LIN {X -0.221,Y -488.600,Z 443.525,A 0.000,B 0.000,C 90.000,E1 274.473} C_DIS
LIN {X -0.021,Y -490.095,Z 443.522,A 0.000,B 0.000,C 90.000,E1 273.955} C_DIS
LIN {X 0.158,Y -491.125,Z 443.519,A 0.000,B 0.000,C 90.000,E1 273.440} C_DIS
LIN {X -0.115,Y -491.790,Z 443.516,A 0.000,B 0.000,C 90.000,E1 272.980} C_DIS
LIN {X 0.083,Y -492.033,Z 443.514,A 0.000,B 0.000,C 90.000,E1 272.465} C_DIS
LIN {X -0.204,Y -491.927,Z 443.511,A 0.000,B 0.000,C 90.000,E1 272.007} C_DIS
LIN {X 0.017,Y -491.436,Z 443.508,A 0.000,B 0.000,C 90.000,E1 271.489} C_DIS
LIN {X 0.222,Y -490.584,Z 443.506,A 0.000,B 0.000,C 90.000,E1 270.974} C_DIS
LIN {X -0.065,Y -489.225,Z 443.503,A 0.000,B 0.000,C 90.000,E1 270.516} C_DIS
LIN {X 0.134,Y -487.368,Z 443.500,A 0.000,B 0.000,C 90.000,E1 270.000} C_DIS
LIN {X -0.162,Y -484.881,Z 443.497,A 0.000,B 0.000,C 90.000,E1 269.542} C_DIS
LIN {X 0.010,Y -481.643,Z 443.495,A 0.000,B 0.000,C 90.000,E1 269.026} C_DIS
LIN {X 0.162,Y -477.508,Z 443.492,A 0.000,B 0.000,C 90.000,E1 268.511} C_DIS
LIN {X -0.011,Y -475.068,Z 443.490,A 0.000,B 0.000,C 90.000,E1 268.282} C_DIS
LIN {X -0.179,Y -469.417,Z 443.488,A 0.000,B 0.000,C 90.000,E1 267.822} C_DIS
LIN {X 0.061,Y -463.154,Z 443.485,A 0.000,B 0.000,C 90.000,E1 267.364} C_DIS
LIN {X -0.087,Y -456.461,Z 443.483,A 0.000,B 0.000,C 90.000,E1 267.020} C_DIS
LIN {X -0.181,Y -449.602,Z 443.482,A 0.000,B 0.000,C 90.000,E1 266.731} C_DIS
LIN {X 0.068,Y -442.526,Z 443.480,A 0.000,B 0.000,C 90.000,E1 266.445} C_DIS
LIN {X -0.215,Y -434.939,Z 443.479,A 0.000,B 0.000,C 90.000,E1 266.274} C_DIS
LIN {X -0.097,Y -426.109,Z 443.478,A 0.000,B 0.000,C 90.000,E1 266.102} C_DIS
LIN {X -0.029,Y -415.201,Z 443.478,A 0.000,B 0.000,C 90.000,E1 265.988} C_DIS
LIN {X 0.157,Y -408.755,Z 443.478,A 0.000,B 0.000,C 90.000,E1 265.931} C_DIS
LIN {X 0.049,Y -180.918,Z 443.477,A 0.000,B 0.000,C 90.000,E1 265.927} C_DIS
LIN {X 0.081,Y -180.842,Z 443.472,A 0.000,B 0.000,C 90.000,E1 264.894} C_DIS
LIN {X -0.022,Y -178.884,Z 443.443,A 0.000,B 0.000,C 90.000,E1 259.690} C_DIS
LIN {X 0.053,Y -175.927,Z 443.414,A 0.000,B 0.000,C 90.000,E1 254.574} C_DIS
LIN {X -0.001,Y -175.367,Z 443.410,A 0.000,B 0.000,C 90.000,E1 253.740} C_DIS
LIN {X 0.058,Y -172.144,Z 443.386,A 0.000,B 0.000,C 90.000,E1 249.444} C_DIS
LIN {X 0.035,Y -171.609,Z 443.381,A 0.000,B 0.000,C 90.000,E1 248.592} C_DIS
LIN {X 0.023,Y -167.831,Z 443.357,A 0.000,B 0.000,C 90.000,E1 244.280} C_DIS
LIN {X 0.040,Y -166.558,Z 443.348,A 0.000,B 0.000,C 90.000,E1 242.538} C_DIS
LIN {X -0.050,Y -162.553,Z 443.323,A 0.000,B 0.000,C 90.000,E1 238.201} C_DIS
LIN {X 0.011,Y -161.231,Z 443.313,A 0.000,B 0.000,C 90.000,E1 236.421} C_DIS
LIN {X 0.045,Y -157.236,Z 443.289,A 0.000,B 0.000,C 90.000,E1 231.984} C_DIS
LIN {X -0.031,Y -155.961,Z 443.279,A 0.000,B 0.000,C 90.000,E1 230.231} C_DIS
LIN {X 0.026,Y -152.214,Z 443.254,A 0.000,B 0.000,C 90.000,E1 225.729} C_DIS
LIN {X 0.048,Y -150.459,Z 443.239,A 0.000,B 0.000,C 90.000,E1 223.014} C_DIS
LIN {X 0.073,Y -147.184,Z 443.214,A 0.000,B 0.000,C 90.000,E1 218.463} C_DIS
LIN {X 0.039,Y -145.201,Z 443.194,A 0.000,B 0.000,C 90.000,E1 214.818} C_DIS
LIN {X -0.051,Y -142.339,Z 443.163,A 0.000,B 0.000,C 90.000,E1 209.333} C_DIS
LIN {X 0.003,Y -141.727,Z 443.153,A 0.000,B 0.000,C 90.000,E1 207.462} C_DIS
LIN {X -0.015,Y -139.480,Z 443.116,A 0.000,B 0.000,C 90.000,E1 200.972} C_DIS
LIN {X -0.026,Y -138.979,Z 443.101,A 0.000,B 0.000,C 90.000,E1 198.181} C_DIS
LIN {X -0.041,Y -138.332,Z 443.054,A 0.000,B 0.000,C 90.000,E1 189.782} C_DIS
LIN {X -0.040,Y -139.429,Z 443.008,A 0.000,B 0.000,C 90.000,E1 181.375} C_DIS
LIN {X 0.013,Y -141.356,Z 442.971,A 0.000,B 0.000,C 90.000,E1 174.837} C_DIS
LIN {X -0.011,Y -142.710,Z 442.956,A 0.000,B 0.000,C 90.000,E1 172.064} C_DIS
LIN {X -0.052,Y -145.085,Z 442.930,A 0.000,B 0.000,C 90.000,E1 167.465} C_DIS
LIN {X -0.056,Y -147.708,Z 442.910,A 0.000,B 0.000,C 90.000,E1 163.795} C_DIS
LIN {X 0.027,Y -150.364,Z 442.890,A 0.000,B 0.000,C 90.000,E1 160.115} C_DIS
LIN {X 0.045,Y -153.790,Z 442.869,A 0.000,B 0.000,C 90.000,E1 156.485} C_DIS
LIN {X -0.035,Y -157.202,Z 442.849,A 0.000,B 0.000,C 90.000,E1 152.922} C_DIS
LIN {X 0.048,Y -161.364,Z 442.830,A 0.000,B 0.000,C 90.000,E1 149.331} C_DIS
LIN {X 0.059,Y -165.566,Z 442.810,A 0.000,B 0.000,C 90.000,E1 145.801} C_DIS
LIN {X -0.058,Y -170.484,Z 442.791,A 0.000,B 0.000,C 90.000,E1 142.351} C_DIS
LIN {X 0.091,Y -175.364,Z 442.772,A 0.000,B 0.000,C 90.000,E1 138.852} C_DIS
LIN {X -0.046,Y -180.989,Z 442.753,A 0.000,B 0.000,C 90.000,E1 135.486} C_DIS
LIN {X 0.078,Y -186.416,Z 442.734,A 0.000,B 0.000,C 90.000,E1 132.081} C_DIS
LIN {X -0.120,Y -191.043,Z 442.720,A 0.000,B 0.000,C 90.000,E1 129.644} C_DIS
LIN {X 0.051,Y -195.459,Z 442.706,A 0.000,B 0.000,C 90.000,E1 127.030} C_DIS
LIN {X 0.043,Y -293.930,Z 442.706,A 0.000,B 0.000,C 90.000,E1 127.030} C_DIS
LIN {X 0.008,Y -295.930,Z 442.706,A 0.000,B 0.000,C 90.000,E1 126.996} C_DIS
LIN {X -0.031,Y -301.628,Z 442.704,A 0.000,B 0.000,C 90.000,E1 126.664} C_DIS
LIN {X 0.110,Y -304.652,Z 442.702,A 0.000,B 0.000,C 90.000,E1 126.297} C_DIS
LIN {X -0.010,Y -306.653,Z 442.700,A 0.000,B 0.000,C 90.000,E1 126.011} C_DIS
LIN {X -0.131,Y -308.223,Z 442.698,A 0.000,B 0.000,C 90.000,E1 125.724} C_DIS
LIN {X -0.098,Y -309.544,Z 442.697,A 0.000,B 0.000,C 90.000,E1 125.391} C_DIS
LIN {X 0.094,Y -321.296,Z 442.677,A 0.000,B 0.000,C 90.000,E1 121.799} C_DIS
LIN {X 0.084,Y -332.295,Z 442.661,A 0.000,B 0.000,C 90.000,E1 118.949} C_DIS
LIN {X 0.060,Y -344.702,Z 442.645,A 0.000,B 0.000,C 90.000,E1 116.155} C_DIS
LIN {X 0.063,Y -357.000,Z 442.632,A 0.000,B 0.000,C 90.000,E1 113.718} C_DIS
LIN {X -0.086,Y -370.586,Z 442.619,A 0.000,B 0.000,C 90.000,E1 111.354} C_DIS
LIN {X -0.177,Y -385.559,Z 442.606,A 0.000,B 0.000,C 90.000,E1 109.033} C_DIS
LIN {X -0.027,Y -402.029,Z 442.593,A 0.000,B 0.000,C 90.000,E1 106.732} C_DIS
LIN {X -0.210,Y -420.117,Z 442.581,A 0.000,B 0.000,C 90.000,E1 104.537} C_DIS
LIN {X 0.085,Y -439.785,Z 442.569,A 0.000,B 0.000,C 90.000,E1 102.355} C_DIS
LIN {X 0.197,Y -460.169,Z 442.558,A 0.000,B 0.000,C 90.000,E1 100.366} C_DIS
LIN {X 0.203,Y -483.699,Z 442.546,A 0.000,B 0.000,C 90.000,E1 98.341} C_DIS
LIN {X -0.104,Y -485.940,Z 442.545,A 0.000,B 0.000,C 90.000,E1 98.163} C_DIS
LIN {X -0.199,Y -487.805,Z 442.544,A 0.000,B 0.000,C 90.000,E1 97.936} C_DIS
LIN {X -0.225,Y -489.220,Z 442.543,A 0.000,B 0.000,C 90.000,E1 97.701} C_DIS
LIN {X -0.015,Y -491.110,Z 442.540,A 0.000,B 0.000,C 90.000,E1 97.182} C_DIS
LIN {X 0.204,Y -491.879,Z 442.537,A 0.000,B 0.000,C 90.000,E1 96.663} C_DIS
LIN {X -0.053,Y -491.656,Z 442.534,A 0.000,B 0.000,C 90.000,E1 96.201} C_DIS
LIN {X 0.181,Y -490.409,Z 442.532,A 0.000,B 0.000,C 90.000,E1 95.682} C_DIS
LIN {X 0.031,Y -489.338,Z 442.530,A 0.000,B 0.000,C 90.000,E1 95.454} C_DIS
LIN {X -0.074,Y -487.898,Z 442.529,A 0.000,B 0.000,C 90.000,E1 95.220} C_DIS
LIN {X -0.182,Y -480.142,Z 442.523,A 0.000,B 0.000,C 90.000,E1 94.245} C_DIS
LIN {X 0.089,Y -462.283,Z 442.511,A 0.000,B 0.000,C 90.000,E1 91.949} C_DIS
LIN {X -0.076,Y -449.413,Z 442.501,A 0.000,B 0.000,C 90.000,E1 90.172} C_DIS
LIN {X -0.147,Y -434.329,Z 442.488,A 0.000,B 0.000,C 90.000,E1 87.822} C_DIS
LIN {X 0.087,Y -416.543,Z 442.471,A 0.000,B 0.000,C 90.000,E1 84.837} C_DIS
LIN {X 0.027,Y -404.185,Z 442.459,A 0.000,B 0.000,C 90.000,E1 82.648} C_DIS
LIN {X 0.110,Y -393.487,Z 442.448,A 0.000,B 0.000,C 90.000,E1 80.679} C_DIS
LIN {X 0.068,Y -381.309,Z 442.436,A 0.000,B 0.000,C 90.000,E1 78.409} C_DIS
LIN {X -0.020,Y -368.027,Z 442.421,A 0.000,B 0.000,C 90.000,E1 75.811} C_DIS
LIN {X 0.040,Y -354.202,Z 442.405,A 0.000,B 0.000,C 90.000,E1 72.834} C_DIS
LIN {X -0.103,Y -340.320,Z 442.386,A 0.000,B 0.000,C 90.000,E1 69.518} C_DIS
LIN {X -0.154,Y -330.784,Z 442.372,A 0.000,B 0.000,C 90.000,E1 67.050} C_DIS
LIN {X -0.177,Y -321.387,Z 442.358,A 0.000,B 0.000,C 90.000,E1 64.537} C_DIS
LIN {X -0.092,Y -311.159,Z 442.342,A 0.000,B 0.000,C 90.000,E1 61.641} C_DIS
LIN {X 0.117,Y -302.250,Z 442.328,A 0.000,B 0.000,C 90.000,E1 58.997} C_DIS
LIN {X -0.061,Y -291.852,Z 442.310,A 0.000,B 0.000,C 90.000,E1 55.722} C_DIS
LIN {X -0.056,Y -282.281,Z 442.291,A 0.000,B 0.000,C 90.000,E1 52.351} C_DIS
LIN {X 0.067,Y -276.551,Z 442.279,A 0.000,B 0.000,C 90.000,E1 50.275} C_DIS
LIN {X -0.127,Y -270.634,Z 442.268,A 0.000,B 0.000,C 90.000,E1 48.243} C_DIS
LIN {X -0.068,Y -264.485,Z 442.256,A 0.000,B 0.000,C 90.000,E1 46.134} C_DIS
LIN {X -0.131,Y -258.184,Z 442.244,A 0.000,B 0.000,C 90.000,E1 44.028} C_DIS
LIN {X 0.056,Y -251.742,Z 442.233,A 0.000,B 0.000,C 90.000,E1 41.838} C_DIS
LIN {X -0.041,Y -243.162,Z 442.216,A 0.000,B 0.000,C 90.000,E1 38.955} C_DIS
LIN {X 0.047,Y -233.016,Z 442.196,A 0.000,B 0.000,C 90.000,E1 35.231} C_DIS
LIN {X 0.056,Y -225.712,Z 442.179,A 0.000,B 0.000,C 90.000,E1 32.212} C_DIS
LIN {X 0.035,Y -219.253,Z 442.162,A 0.000,B 0.000,C 90.000,E1 29.155} C_DIS
LIN {X 0.030,Y -213.522,Z 442.145,A 0.000,B 0.000,C 90.000,E1 26.052} C_DIS
LIN {X -0.085,Y -207.363,Z 442.123,A 0.000,B 0.000,C 90.000,E1 22.153} C_DIS
LIN {X 0.069,Y -202.138,Z 442.101,A 0.000,B 0.000,C 90.000,E1 18.127} C_DIS
LIN {X 0.001,Y -197.867,Z 442.078,A 0.000,B 0.000,C 90.000,E1 14.120} C_DIS
LIN {X -0.081,Y -193.976,Z 442.051,A 0.000,B 0.000,C 90.000,E1 9.265} C_DIS
LIN {X -0.053,Y -190.959,Z 442.015,A 0.000,B 0.000,C 90.000,E1 2.694} C_DIS
LIN {X 0.013,Y -191.662,Z 441.961,A 0.000,B 0.000,C 90.000,E1 352.932} C_DIS
LIN {X 0.050,Y -194.824,Z 441.929,A 0.000,B 0.000,C 90.000,E1 347.173} C_DIS
LIN {X -0.037,Y -198.936,Z 441.902,A 0.000,B 0.000,C 90.000,E1 342.308} C_DIS
LIN {X -0.092,Y -203.435,Z 441.879,A 0.000,B 0.000,C 90.000,E1 338.284} C_DIS
LIN {X -0.075,Y -209.043,Z 441.857,A 0.000,B 0.000,C 90.000,E1 334.280} C_DIS
LIN {X -0.081,Y -215.362,Z 441.835,A 0.000,B 0.000,C 90.000,E1 330.333} C_DIS
LIN {X -0.014,Y -222.210,Z 441.813,A 0.000,B 0.000,C 90.000,E1 326.421} C_DIS
LIN {X 0.093,Y -229.806,Z 441.792,A 0.000,B 0.000,C 90.000,E1 322.557} C_DIS
LIN {X 0.139,Y -238.270,Z 441.771,A 0.000,B 0.000,C 90.000,E1 318.771} C_DIS
LIN {X -0.097,Y -246.873,Z 441.753,A 0.000,B 0.000,C 90.000,E1 315.486} C_DIS
LIN {X -0.078,Y -256.744,Z 441.734,A 0.000,B 0.000,C 90.000,E1 312.204} C_DIS
LIN {X -0.069,Y -267.737,Z 441.717,A 0.000,B 0.000,C 90.000,E1 308.991} C_DIS
LIN {X 0.143,Y -279.758,Z 441.699,A 0.000,B 0.000,C 90.000,E1 305.804} C_DIS
LIN {X 0.056,Y -292.507,Z 441.682,A 0.000,B 0.000,C 90.000,E1 302.752} C_DIS
LIN {X 0.136,Y -307.604,Z 441.664,A 0.000,B 0.000,C 90.000,E1 299.411} C_DIS
LIN {X 0.103,Y -320.663,Z 441.649,A 0.000,B 0.000,C 90.000,E1 296.821} C_DIS
LIN {X -0.095,Y -338.641,Z 441.632,A 0.000,B 0.000,C 90.000,E1 293.695} C_DIS
LIN {X -0.036,Y -354.873,Z 441.618,A 0.000,B 0.000,C 90.000,E1 291.227} C_DIS
LIN {X -0.057,Y -374.926,Z 441.603,A 0.000,B 0.000,C 90.000,E1 288.544} C_DIS
LIN {X 0.108,Y -394.293,Z 441.590,A 0.000,B 0.000,C 90.000,E1 286.205} C_DIS
LIN {X -0.009,Y -414.495,Z 441.578,A 0.000,B 0.000,C 90.000,E1 284.120} C_DIS
LIN {X -0.076,Y -429.766,Z 441.570,A 0.000,B 0.000,C 90.000,E1 282.647} C_DIS
LIN {X -0.049,Y -437.275,Z 441.566,A 0.000,B 0.000,C 90.000,E1 281.883} C_DIS
LIN {X -0.057,Y -446.995,Z 441.560,A 0.000,B 0.000,C 90.000,E1 280.838} C_DIS
LIN {X 0.214,Y -453.820,Z 441.556,A 0.000,B 0.000,C 90.000,E1 280.018} C_DIS
LIN {X 0.023,Y -460.130,Z 441.551,A 0.000,B 0.000,C 90.000,E1 279.265} C_DIS
LIN {X -0.123,Y -465.964,Z 441.547,A 0.000,B 0.000,C 90.000,E1 278.511} C_DIS
LIN {X -0.214,Y -471.253,Z 441.543,A 0.000,B 0.000,C 90.000,E1 277.757} C_DIS
LIN {X 0.003,Y -477.535,Z 441.537,A 0.000,B 0.000,C 90.000,E1 276.720} C_DIS
LIN {X 0.004,Y -481.829,Z 441.533,A 0.000,B 0.000,C 90.000,E1 275.967} C_DIS
LIN {X -0.005,Y -485.537,Z 441.529,A 0.000,B 0.000,C 90.000,E1 275.220} C_DIS
LIN {X 0.017,Y -488.538,Z 441.525,A 0.000,B 0.000,C 90.000,E1 274.473} C_DIS
LIN {X 0.217,Y -490.028,Z 441.522,A 0.000,B 0.000,C 90.000,E1 273.955} C_DIS
LIN {X -0.095,Y -491.088,Z 441.519,A 0.000,B 0.000,C 90.000,E1 273.498} C_DIS
LIN {X 0.122,Y -491.751,Z 441.517,A 0.000,B 0.000,C 90.000,E1 272.980} C_DIS
LIN {X -0.171,Y -492.032,Z 441.514,A 0.000,B 0.000,C 90.000,E1 272.522} C_DIS
LIN {X 0.033,Y -491.961,Z 441.511,A 0.000,B 0.000,C 90.000,E1 272.007} C_DIS
LIN {X -0.237,Y -491.525,Z 441.508,A 0.000,B 0.000,C 90.000,E1 271.547} C_DIS
LIN {X -0.031,Y -490.643,Z 441.506,A 0.000,B 0.000,C 90.000,E1 271.031} C_DIS
LIN {X 0.172,Y -489.327,Z 441.503,A 0.000,B 0.000,C 90.000,E1 270.516} C_DIS
LIN {X -0.117,Y -487.469,Z 441.500,A 0.000,B 0.000,C 90.000,E1 270.057} C_DIS
LIN {X 0.222,Y -486.381,Z 441.499,A 0.000,B 0.000,C 90.000,E1 269.771} C_DIS
LIN {X -0.082,Y -483.585,Z 441.496,A 0.000,B 0.000,C 90.000,E1 269.312} C_DIS
LIN {X 0.081,Y -480.000,Z 441.493,A 0.000,B 0.000,C 90.000,E1 268.797} C_DIS
LIN {X 0.222,Y -475.473,Z 441.491,A 0.000,B 0.000,C 90.000,E1 268.282} C_DIS
LIN {X 0.065,Y -472.744,Z 441.489,A 0.000,B 0.000,C 90.000,E1 268.051} C_DIS
LIN {X -0.005,Y -466.708,Z 441.487,A 0.000,B 0.000,C 90.000,E1 267.593} C_DIS
LIN {X 0.210,Y -463.599,Z 441.486,A 0.000,B 0.000,C 90.000,E1 267.364} C_DIS
LIN {X 0.019,Y -456.902,Z 441.483,A 0.000,B 0.000,C 90.000,E1 267.020} C_DIS
LIN {X -0.085,Y -450.003,Z 441.482,A 0.000,B 0.000,C 90.000,E1 266.731} C_DIS
LIN {X 0.158,Y -442.978,Z 441.480,A 0.000,B 0.000,C 90.000,E1 266.445} C_DIS
LIN {X -0.148,Y -435.436,Z 441.479,A 0.000,B 0.000,C 90.000,E1 266.274} C_DIS
LIN {X -0.055,Y -426.538,Z 441.478,A 0.000,B 0.000,C 90.000,E1 266.102} C_DIS
LIN {X -0.149,Y -412.752,Z 441.478,A 0.000,B 0.000,C 90.000,E1 265.988} C_DIS
LIN {X 0.139,Y -407.658,Z 441.477,A 0.000,B 0.000,C 90.000,E1 265.927} C_DIS
LIN {X 0.040,Y -180.918,Z 441.477,A 0.000,B 0.000,C 90.000,E1 265.927} C_DIS
LIN {X -0.050,Y -180.873,Z 441.473,A 0.000,B 0.000,C 90.000,E1 265.065} C_DIS
LIN {X 0.007,Y -178.989,Z 441.444,A 0.000,B 0.000,C 90.000,E1 259.982} C_DIS
LIN {X 0.019,Y -177.971,Z 441.435,A 0.000,B 0.000,C 90.000,E1 258.285} C_DIS
LIN {X 0.037,Y -175.615,Z 441.411,A 0.000,B 0.000,C 90.000,E1 254.031} C_DIS
LIN {X 0.049,Y -172.336,Z 441.388,A 0.000,B 0.000,C 90.000,E1 249.752} C_DIS
LIN {X 0.028,Y -171.813,Z 441.383,A 0.000,B 0.000,C 90.000,E1 248.901} C_DIS
LIN {X 0.036,Y -170.277,Z 441.373,A 0.000,B 0.000,C 90.000,E1 247.177} C_DIS
LIN {X -0.029,Y -166.818,Z 441.349,A 0.000,B 0.000,C 90.000,E1 242.871} C_DIS
LIN {X 0.028,Y -162.800,Z 441.325,A 0.000,B 0.000,C 90.000,E1 238.486} C_DIS
LIN {X -0.046,Y -161.487,Z 441.315,A 0.000,B 0.000,C 90.000,E1 236.755} C_DIS
LIN {X 0.004,Y -157.483,Z 441.291,A 0.000,B 0.000,C 90.000,E1 232.316} C_DIS
LIN {X 0.061,Y -155.500,Z 441.276,A 0.000,B 0.000,C 90.000,E1 229.622} C_DIS
LIN {X -0.007,Y -151.804,Z 441.251,A 0.000,B 0.000,C 90.000,E1 225.162} C_DIS
LIN {X 0.006,Y -150.015,Z 441.236,A 0.000,B 0.000,C 90.000,E1 222.447} C_DIS
LIN {X 0.036,Y -146.840,Z 441.211,A 0.000,B 0.000,C 90.000,E1 217.890} C_DIS
LIN {X 0.023,Y -145.420,Z 441.195,A 0.000,B 0.000,C 90.000,E1 215.152} C_DIS
LIN {X -0.065,Y -142.848,Z 441.170,A 0.000,B 0.000,C 90.000,E1 210.590} C_DIS
LIN {X -0.012,Y -141.462,Z 441.149,A 0.000,B 0.000,C 90.000,E1 206.873} C_DIS
LIN {X -0.022,Y -139.376,Z 441.113,A 0.000,B 0.000,C 90.000,E1 200.375} C_DIS
LIN {X -0.030,Y -138.826,Z 441.098,A 0.000,B 0.000,C 90.000,E1 197.583} C_DIS
LIN {X 0.058,Y -138.353,Z 441.056,A 0.000,B 0.000,C 90.000,E1 190.074} C_DIS
LIN {X 0.031,Y -139.530,Z 441.004,A 0.000,B 0.000,C 90.000,E1 180.745} C_DIS
LIN {X -0.016,Y -141.208,Z 440.973,A 0.000,B 0.000,C 90.000,E1 175.179} C_DIS
LIN {X -0.057,Y -142.583,Z 440.958,A 0.000,B 0.000,C 90.000,E1 172.413} C_DIS
LIN {X 0.039,Y -144.878,Z 440.932,A 0.000,B 0.000,C 90.000,E1 167.757} C_DIS
LIN {X -0.007,Y -147.505,Z 440.912,A 0.000,B 0.000,C 90.000,E1 164.102} C_DIS
LIN {X 0.068,Y -150.097,Z 440.891,A 0.000,B 0.000,C 90.000,E1 160.423} C_DIS
LIN {X 0.080,Y -153.452,Z 440.871,A 0.000,B 0.000,C 90.000,E1 156.794} C_DIS
LIN {X -0.068,Y -157.815,Z 440.846,A 0.000,B 0.000,C 90.000,E1 152.359} C_DIS
LIN {X -0.036,Y -162.098,Z 440.827,A 0.000,B 0.000,C 90.000,E1 148.791} C_DIS
LIN {X -0.011,Y -166.297,Z 440.807,A 0.000,B 0.000,C 90.000,E1 145.261} C_DIS
LIN {X -0.015,Y -171.315,Z 440.788,A 0.000,B 0.000,C 90.000,E1 141.778} C_DIS
LIN {X 0.020,Y -176.213,Z 440.768,A 0.000,B 0.000,C 90.000,E1 138.324} C_DIS
LIN {X -0.115,Y -180.491,Z 440.754,A 0.000,B 0.000,C 90.000,E1 135.810} C_DIS
LIN {X -0.004,Y -185.894,Z 440.736,A 0.000,B 0.000,C 90.000,E1 132.405} C_DIS
LIN {X 0.057,Y -190.521,Z 440.722,A 0.000,B 0.000,C 90.000,E1 129.886} C_DIS
LIN {X -0.017,Y -195.559,Z 440.706,A 0.000,B 0.000,C 90.000,E1 126.996} C_DIS
LIN {X -0.060,Y -293.877,Z 440.705,A 0.000,B 0.000,C 90.000,E1 126.996} C_DIS
LIN {X 0.106,Y -294.873,Z 440.705,A 0.000,B 0.000,C 90.000,E1 126.950} C_DIS
LIN {X 0.001,Y -299.336,Z 440.704,A 0.000,B 0.000,C 90.000,E1 126.790} C_DIS
LIN {X 0.136,Y -301.695,Z 440.703,A 0.000,B 0.000,C 90.000,E1 126.583} C_DIS
LIN {X -0.087,Y -305.558,Z 440.701,A 0.000,B 0.000,C 90.000,E1 126.171} C_DIS
LIN {X 0.165,Y -307.445,Z 440.699,A 0.000,B 0.000,C 90.000,E1 125.804} C_DIS
LIN {X -0.013,Y -308.929,Z 440.697,A 0.000,B 0.000,C 90.000,E1 125.518} C_DIS
LIN {X -0.016,Y -311.140,Z 440.694,A 0.000,B 0.000,C 90.000,E1 124.865} C_DIS
LIN {X -0.194,Y -321.921,Z 440.676,A 0.000,B 0.000,C 90.000,E1 121.671} C_DIS
LIN {X -0.194,Y -333.004,Z 440.660,A 0.000,B 0.000,C 90.000,E1 118.821} C_DIS
LIN {X 0.103,Y -345.502,Z 440.644,A 0.000,B 0.000,C 90.000,E1 115.976} C_DIS
LIN {X -0.050,Y -357.886,Z 440.631,A 0.000,B 0.000,C 90.000,E1 113.567} C_DIS
LIN {X 0.014,Y -371.566,Z 440.618,A 0.000,B 0.000,C 90.000,E1 111.173} C_DIS
LIN {X -0.047,Y -386.640,Z 440.605,A 0.000,B 0.000,C 90.000,E1 108.852} C_DIS
LIN {X 0.020,Y -403.220,Z 440.592,A 0.000,B 0.000,C 90.000,E1 106.567} C_DIS
LIN {X -0.013,Y -421.426,Z 440.580,A 0.000,B 0.000,C 90.000,E1 104.356} C_DIS
LIN {X -0.170,Y -441.178,Z 440.568,A 0.000,B 0.000,C 90.000,E1 102.243} C_DIS
LIN {X 0.032,Y -461.601,Z 440.557,A 0.000,B 0.000,C 90.000,E1 100.254} C_DIS
LIN {X 0.206,Y -485.047,Z 440.546,A 0.000,B 0.000,C 90.000,E1 98.219} C_DIS
LIN {X -0.160,Y -486.986,Z 440.545,A 0.000,B 0.000,C 90.000,E1 98.049} C_DIS
LIN {X 0.212,Y -488.696,Z 440.543,A 0.000,B 0.000,C 90.000,E1 97.757} C_DIS
LIN {X 0.034,Y -489.978,Z 440.542,A 0.000,B 0.000,C 90.000,E1 97.530} C_DIS
LIN {X -0.236,Y -491.561,Z 440.539,A 0.000,B 0.000,C 90.000,E1 97.068} C_DIS
LIN {X -0.010,Y -492.074,Z 440.536,A 0.000,B 0.000,C 90.000,E1 96.549} C_DIS
LIN {X -0.264,Y -491.602,Z 440.534,A 0.000,B 0.000,C 90.000,E1 96.087} C_DIS
LIN {X -0.027,Y -490.069,Z 440.531,A 0.000,B 0.000,C 90.000,E1 95.568} C_DIS
LIN {X -0.132,Y -488.822,Z 440.530,A 0.000,B 0.000,C 90.000,E1 95.334} C_DIS
LIN {X 0.048,Y -485.252,Z 440.527,A 0.000,B 0.000,C 90.000,E1 94.821} C_DIS
LIN {X 0.070,Y -473.324,Z 440.519,A 0.000,B 0.000,C 90.000,E1 93.326} C_DIS
LIN {X 0.158,Y -455.848,Z 440.506,A 0.000,B 0.000,C 90.000,E1 91.031} C_DIS
LIN {X -0.146,Y -443.590,Z 440.496,A 0.000,B 0.000,C 90.000,E1 89.255} C_DIS
LIN {X -0.080,Y -430.295,Z 440.484,A 0.000,B 0.000,C 90.000,E1 87.135} C_DIS
LIN {X 0.046,Y -412.781,Z 440.468,A 0.000,B 0.000,C 90.000,E1 84.147} C_DIS
LIN {X -0.050,Y -400.468,Z 440.455,A 0.000,B 0.000,C 90.000,E1 81.951} C_DIS
LIN {X -0.099,Y -391.322,Z 440.446,A 0.000,B 0.000,C 90.000,E1 80.274} C_DIS
LIN {X -0.144,Y -380.705,Z 440.435,A 0.000,B 0.000,C 90.000,E1 78.285} C_DIS
LIN {X 0.035,Y -367.479,Z 440.420,A 0.000,B 0.000,C 90.000,E1 75.644} C_DIS
LIN {X 0.062,Y -353.719,Z 440.404,A 0.000,B 0.000,C 90.000,E1 72.670} C_DIS
LIN {X -0.003,Y -341.078,Z 440.387,A 0.000,B 0.000,C 90.000,E1 69.645} C_DIS
LIN {X -0.065,Y -330.288,Z 440.371,A 0.000,B 0.000,C 90.000,E1 66.869} C_DIS
LIN {X -0.023,Y -319.705,Z 440.356,A 0.000,B 0.000,C 90.000,E1 64.024} C_DIS
LIN {X 0.006,Y -309.500,Z 440.340,A 0.000,B 0.000,C 90.000,E1 61.129} C_DIS
LIN {X -0.025,Y -297.455,Z 440.320,A 0.000,B 0.000,C 90.000,E1 57.533} C_DIS
LIN {X -0.020,Y -287.464,Z 440.301,A 0.000,B 0.000,C 90.000,E1 54.196} C_DIS
LIN {X 0.110,Y -279.901,Z 440.286,A 0.000,B 0.000,C 90.000,E1 51.457} C_DIS
LIN {X 0.186,Y -274.101,Z 440.275,A 0.000,B 0.000,C 90.000,E1 49.380} C_DIS
LIN {X 0.123,Y -268.104,Z 440.263,A 0.000,B 0.000,C 90.000,E1 47.310} C_DIS
LIN {X -0.061,Y -261.877,Z 440.251,A 0.000,B 0.000,C 90.000,E1 45.243} C_DIS
LIN {X 0.014,Y -255.544,Z 440.239,A 0.000,B 0.000,C 90.000,E1 43.095} C_DIS
LIN {X -0.017,Y -249.062,Z 440.227,A 0.000,B 0.000,C 90.000,E1 40.943} C_DIS
LIN {X -0.010,Y -238.525,Z 440.207,A 0.000,B 0.000,C 90.000,E1 37.282} C_DIS
LIN {X 0.074,Y -230.698,Z 440.191,A 0.000,B 0.000,C 90.000,E1 34.278} C_DIS
LIN {X 0.027,Y -223.634,Z 440.174,A 0.000,B 0.000,C 90.000,E1 31.258} C_DIS
LIN {X 0.037,Y -217.402,Z 440.157,A 0.000,B 0.000,C 90.000,E1 28.180} C_DIS
LIN {X -0.016,Y -211.891,Z 440.139,A 0.000,B 0.000,C 90.000,E1 25.079} C_DIS
LIN {X 0.111,Y -205.969,Z 440.117,A 0.000,B 0.000,C 90.000,E1 21.099} C_DIS
LIN {X -0.047,Y -200.912,Z 440.095,A 0.000,B 0.000,C 90.000,E1 17.149} C_DIS
LIN {X -0.070,Y -196.901,Z 440.073,A 0.000,B 0.000,C 90.000,E1 13.119} C_DIS
LIN {X -0.006,Y -193.787,Z 440.050,A 0.000,B 0.000,C 90.000,E1 9.029} C_DIS
LIN {X -0.009,Y -190.824,Z 440.014,A 0.000,B 0.000,C 90.000,E1 2.465} C_DIS
LIN {X 0.007,Y -191.536,Z 439.961,A 0.000,B 0.000,C 90.000,E1 352.932} C_DIS
LIN {X 0.039,Y -194.677,Z 439.929,A 0.000,B 0.000,C 90.000,E1 347.173} C_DIS
LIN {X -0.053,Y -198.790,Z 439.902,A 0.000,B 0.000,C 90.000,E1 342.308} C_DIS
LIN {X 0.075,Y -203.286,Z 439.879,A 0.000,B 0.000,C 90.000,E1 338.230} C_DIS
LIN {X -0.101,Y -208.887,Z 439.857,A 0.000,B 0.000,C 90.000,E1 334.280} C_DIS
LIN {X -0.113,Y -215.218,Z 439.835,A 0.000,B 0.000,C 90.000,E1 330.333} C_DIS
LIN {X -0.051,Y -222.064,Z 439.813,A 0.000,B 0.000,C 90.000,E1 326.421} C_DIS
LIN {X 0.049,Y -229.681,Z 439.792,A 0.000,B 0.000,C 90.000,E1 322.557} C_DIS
LIN {X 0.089,Y -238.145,Z 439.771,A 0.000,B 0.000,C 90.000,E1 318.771} C_DIS
LIN {X 0.023,Y -246.774,Z 439.753,A 0.000,B 0.000,C 90.000,E1 315.445} C_DIS
LIN {X 0.031,Y -255.473,Z 439.736,A 0.000,B 0.000,C 90.000,E1 312.528} C_DIS
LIN {X -0.030,Y -266.368,Z 439.718,A 0.000,B 0.000,C 90.000,E1 309.322} C_DIS
LIN {X -0.027,Y -278.304,Z 439.701,A 0.000,B 0.000,C 90.000,E1 306.171} C_DIS
LIN {X 0.023,Y -289.574,Z 439.686,A 0.000,B 0.000,C 90.000,E1 303.420} C_DIS
LIN {X 0.002,Y -304.456,Z 439.667,A 0.000,B 0.000,C 90.000,E1 300.079} C_DIS
LIN {X 0.094,Y -318.955,Z 439.651,A 0.000,B 0.000,C 90.000,E1 297.129} C_DIS
LIN {X 0.143,Y -336.750,Z 439.633,A 0.000,B 0.000,C 90.000,E1 293.951} C_DIS
LIN {X -0.161,Y -352.820,Z 439.620,A 0.000,B 0.000,C 90.000,E1 291.535} C_DIS
LIN {X -0.119,Y -372.702,Z 439.605,A 0.000,B 0.000,C 90.000,E1 288.833} C_DIS
LIN {X 0.010,Y -394.404,Z 439.590,A 0.000,B 0.000,C 90.000,E1 286.205} C_DIS
LIN {X 0.100,Y -414.930,Z 439.578,A 0.000,B 0.000,C 90.000,E1 284.064} C_DIS
LIN {X -0.061,Y -430.346,Z 439.570,A 0.000,B 0.000,C 90.000,E1 282.591} C_DIS
LIN {X -0.069,Y -437.888,Z 439.566,A 0.000,B 0.000,C 90.000,E1 281.827} C_DIS
LIN {X -0.067,Y -447.605,Z 439.560,A 0.000,B 0.000,C 90.000,E1 280.782} C_DIS
LIN {X 0.212,Y -454.344,Z 439.555,A 0.000,B 0.000,C 90.000,E1 279.962} C_DIS
LIN {X 0.025,Y -460.607,Z 439.551,A 0.000,B 0.000,C 90.000,E1 279.208} C_DIS
LIN {X -0.116,Y -466.377,Z 439.547,A 0.000,B 0.000,C 90.000,E1 278.454} C_DIS
LIN {X 0.108,Y -473.231,Z 439.541,A 0.000,B 0.000,C 90.000,E1 277.409} C_DIS
LIN {X -0.123,Y -479.346,Z 439.536,A 0.000,B 0.000,C 90.000,E1 276.429} C_DIS
LIN {X -0.156,Y -483.413,Z 439.531,A 0.000,B 0.000,C 90.000,E1 275.682} C_DIS
LIN {X -0.152,Y -486.874,Z 439.527,A 0.000,B 0.000,C 90.000,E1 274.935} C_DIS
LIN {X 0.044,Y -488.708,Z 439.525,A 0.000,B 0.000,C 90.000,E1 274.416} C_DIS
LIN {X 0.247,Y -490.153,Z 439.522,A 0.000,B 0.000,C 90.000,E1 273.898} C_DIS
LIN {X -0.064,Y -491.179,Z 439.519,A 0.000,B 0.000,C 90.000,E1 273.440} C_DIS
LIN {X 0.154,Y -491.795,Z 439.516,A 0.000,B 0.000,C 90.000,E1 272.922} C_DIS
LIN {X -0.139,Y -492.060,Z 439.514,A 0.000,B 0.000,C 90.000,E1 272.465} C_DIS
LIN {X 0.066,Y -491.967,Z 439.511,A 0.000,B 0.000,C 90.000,E1 271.949} C_DIS
LIN {X -0.204,Y -491.497,Z 439.508,A 0.000,B 0.000,C 90.000,E1 271.489} C_DIS
LIN {X 0.002,Y -490.555,Z 439.505,A 0.000,B 0.000,C 90.000,E1 270.974} C_DIS
LIN {X 0.205,Y -489.154,Z 439.503,A 0.000,B 0.000,C 90.000,E1 270.458} C_DIS
LIN {X -0.085,Y -487.283,Z 439.500,A 0.000,B 0.000,C 90.000,E1 270.000} C_DIS
LIN {X 0.105,Y -484.778,Z 439.497,A 0.000,B 0.000,C 90.000,E1 269.484} C_DIS
LIN {X -0.207,Y -481.585,Z 439.494,A 0.000,B 0.000,C 90.000,E1 269.026} C_DIS
LIN {X -0.054,Y -477.432,Z 439.492,A 0.000,B 0.000,C 90.000,E1 268.511} C_DIS
LIN {X 0.090,Y -472.224,Z 439.489,A 0.000,B 0.000,C 90.000,E1 267.993} C_DIS
LIN {X 0.060,Y -469.323,Z 439.488,A 0.000,B 0.000,C 90.000,E1 267.764} C_DIS
LIN {X -0.174,Y -462.932,Z 439.485,A 0.000,B 0.000,C 90.000,E1 267.364} C_DIS
LIN {X 0.146,Y -456.190,Z 439.483,A 0.000,B 0.000,C 90.000,E1 266.963} C_DIS
LIN {X 0.079,Y -449.248,Z 439.482,A 0.000,B 0.000,C 90.000,E1 266.674} C_DIS
LIN {X -0.048,Y -442.219,Z 439.480,A 0.000,B 0.000,C 90.000,E1 266.445} C_DIS
LIN {X 0.139,Y -434.669,Z 439.479,A 0.000,B 0.000,C 90.000,E1 266.216} C_DIS
LIN {X -0.160,Y -425.728,Z 439.478,A 0.000,B 0.000,C 90.000,E1 266.102} C_DIS
LIN {X -0.066,Y -414.771,Z 439.478,A 0.000,B 0.000,C 90.000,E1 265.988} C_DIS
LIN {X 0.127,Y -408.830,Z 439.477,A 0.000,B 0.000,C 90.000,E1 265.931} C_DIS
LIN {X 0.037,Y -180.917,Z 439.477,A 0.000,B 0.000,C 90.000,E1 265.927} C_DIS
LIN {X 0.070,Y -180.840,Z 439.472,A 0.000,B 0.000,C 90.000,E1 264.894} C_DIS
LIN {X -0.033,Y -178.882,Z 439.443,A 0.000,B 0.000,C 90.000,E1 259.690} C_DIS
LIN {X 0.042,Y -175.925,Z 439.414,A 0.000,B 0.000,C 90.000,E1 254.574} C_DIS
LIN {X -0.012,Y -175.364,Z 439.410,A 0.000,B 0.000,C 90.000,E1 253.740} C_DIS
LIN {X 0.046,Y -172.142,Z 439.386,A 0.000,B 0.000,C 90.000,E1 249.444} C_DIS
LIN {X 0.023,Y -171.606,Z 439.381,A 0.000,B 0.000,C 90.000,E1 248.592} C_DIS
LIN {X 0.012,Y -167.829,Z 439.357,A 0.000,B 0.000,C 90.000,E1 244.280} C_DIS
LIN {X 0.029,Y -166.555,Z 439.347,A 0.000,B 0.000,C 90.000,E1 242.538} C_DIS
LIN {X -0.060,Y -162.550,Z 439.323,A 0.000,B 0.000,C 90.000,E1 238.201} C_DIS
LIN {X 0.000,Y -161.228,Z 439.313,A 0.000,B 0.000,C 90.000,E1 236.421} C_DIS
LIN {X 0.035,Y -157.234,Z 439.289,A 0.000,B 0.000,C 90.000,E1 231.984} C_DIS
LIN {X 0.057,Y -155.958,Z 439.279,A 0.000,B 0.000,C 90.000,E1 230.194} C_DIS
LIN {X 0.016,Y -152.212,Z 439.254,A 0.000,B 0.000,C 90.000,E1 225.729} C_DIS
LIN {X 0.037,Y -150.455,Z 439.239,A 0.000,B 0.000,C 90.000,E1 223.014} C_DIS
LIN {X 0.064,Y -147.181,Z 439.214,A 0.000,B 0.000,C 90.000,E1 218.463} C_DIS
LIN {X 0.030,Y -145.200,Z 439.194,A 0.000,B 0.000,C 90.000,E1 214.818} C_DIS
LIN {X -0.060,Y -142.337,Z 439.163,A 0.000,B 0.000,C 90.000,E1 209.333} C_DIS
LIN {X -0.007,Y -141.726,Z 439.153,A 0.000,B 0.000,C 90.000,E1 207.462} C_DIS
LIN {X -0.024,Y -139.480,Z 439.116,A 0.000,B 0.000,C 90.000,E1 200.972} C_DIS
LIN {X -0.035,Y -138.979,Z 439.101,A 0.000,B 0.000,C 90.000,E1 198.181} C_DIS
LIN {X -0.050,Y -138.332,Z 439.054,A 0.000,B 0.000,C 90.000,E1 189.782} C_DIS
LIN {X -0.050,Y -139.430,Z 439.008,A 0.000,B 0.000,C 90.000,E1 181.375} C_DIS
LIN {X 0.004,Y -141.358,Z 438.971,A 0.000,B 0.000,C 90.000,E1 174.837} C_DIS
LIN {X -0.021,Y -142.711,Z 438.956,A 0.000,B 0.000,C 90.000,E1 172.064} C_DIS
LIN {X -0.062,Y -145.087,Z 438.930,A 0.000,B 0.000,C 90.000,E1 167.465} C_DIS
LIN {X 0.075,Y -147.711,Z 438.910,A 0.000,B 0.000,C 90.000,E1 163.740} C_DIS
LIN {X 0.017,Y -150.367,Z 438.890,A 0.000,B 0.000,C 90.000,E1 160.115} C_DIS
LIN {X 0.035,Y -153.793,Z 438.869,A 0.000,B 0.000,C 90.000,E1 156.485} C_DIS
LIN {X -0.045,Y -157.206,Z 438.849,A 0.000,B 0.000,C 90.000,E1 152.922} C_DIS
LIN {X 0.037,Y -161.369,Z 438.830,A 0.000,B 0.000,C 90.000,E1 149.331} C_DIS
LIN {X 0.048,Y -165.571,Z 438.810,A 0.000,B 0.000,C 90.000,E1 145.801} C_DIS
LIN {X -0.070,Y -170.490,Z 438.791,A 0.000,B 0.000,C 90.000,E1 142.351} C_DIS
LIN {X 0.080,Y -175.370,Z 438.772,A 0.000,B 0.000,C 90.000,E1 138.852} C_DIS
LIN {X -0.057,Y -180.995,Z 438.753,A 0.000,B 0.000,C 90.000,E1 135.486} C_DIS
LIN {X 0.067,Y -186.422,Z 438.734,A 0.000,B 0.000,C 90.000,E1 132.081} C_DIS
LIN {X 0.015,Y -191.049,Z 438.720,A 0.000,B 0.000,C 90.000,E1 129.600} C_DIS
LIN {X -0.047,Y -195.661,Z 438.705,A 0.000,B 0.000,C 90.000,E1 126.950} C_DIS
LIN {X -0.123,Y -294.241,Z 438.705,A 0.000,B 0.000,C 90.000,E1 126.950} C_DIS
LIN {X -0.086,Y -298.827,Z 438.704,A 0.000,B 0.000,C 90.000,E1 126.790} C_DIS
LIN {X -0.048,Y -301.062,Z 438.703,A 0.000,B 0.000,C 90.000,E1 126.629} C_DIS
LIN {X 0.092,Y -304.108,Z 438.702,A 0.000,B 0.000,C 90.000,E1 126.297} C_DIS
LIN {X 0.119,Y -307.762,Z 438.699,A 0.000,B 0.000,C 90.000,E1 125.724} C_DIS
LIN {X -0.106,Y -309.248,Z 438.697,A 0.000,B 0.000,C 90.000,E1 125.438} C_DIS
LIN {X -0.075,Y -312.437,Z 438.691,A 0.000,B 0.000,C 90.000,E1 124.452} C_DIS
LIN {X -0.026,Y -322.254,Z 438.675,A 0.000,B 0.000,C 90.000,E1 121.544} C_DIS
LIN {X -0.012,Y -333.386,Z 438.659,A 0.000,B 0.000,C 90.000,E1 118.693} C_DIS
LIN {X -0.003,Y -345.931,Z 438.644,A 0.000,B 0.000,C 90.000,E1 115.899} C_DIS
LIN {X 0.030,Y -358.363,Z 438.630,A 0.000,B 0.000,C 90.000,E1 113.462} C_DIS
LIN {X -0.092,Y -372.094,Z 438.617,A 0.000,B 0.000,C 90.000,E1 111.099} C_DIS
LIN {X -0.152,Y -387.222,Z 438.604,A 0.000,B 0.000,C 90.000,E1 108.779} C_DIS
LIN {X -0.085,Y -403.861,Z 438.592,A 0.000,B 0.000,C 90.000,E1 106.496} C_DIS
LIN {X 0.187,Y -422.132,Z 438.579,A 0.000,B 0.000,C 90.000,E1 104.245} C_DIS
LIN {X 0.191,Y -441.909,Z 438.567,A 0.000,B 0.000,C 90.000,E1 102.119} C_DIS
LIN {X -0.084,Y -462.352,Z 438.557,A 0.000,B 0.000,C 90.000,E1 100.197} C_DIS
LIN {X -0.048,Y -483.304,Z 438.547,A 0.000,B 0.000,C 90.000,E1 98.398} C_DIS
LIN {X 0.123,Y -485.722,Z 438.545,A 0.000,B 0.000,C 90.000,E1 98.163} C_DIS
LIN {X 0.121,Y -487.643,Z 438.544,A 0.000,B 0.000,C 90.000,E1 97.936} C_DIS
LIN {X 0.186,Y -489.114,Z 438.543,A 0.000,B 0.000,C 90.000,E1 97.701} C_DIS
LIN {X 0.079,Y -490.327,Z 438.542,A 0.000,B 0.000,C 90.000,E1 97.466} C_DIS
LIN {X -0.091,Y -491.212,Z 438.540,A 0.000,B 0.000,C 90.000,E1 97.239} C_DIS
LIN {X 0.134,Y -492.146,Z 438.537,A 0.000,B 0.000,C 90.000,E1 96.720} C_DIS
LIN {X -0.123,Y -492.082,Z 438.535,A 0.000,B 0.000,C 90.000,E1 96.258} C_DIS
LIN {X 0.113,Y -491.008,Z 438.532,A 0.000,B 0.000,C 90.000,E1 95.739} C_DIS
LIN {X -0.037,Y -490.043,Z 438.531,A 0.000,B 0.000,C 90.000,E1 95.511} C_DIS
LIN {X -0.140,Y -488.730,Z 438.529,A 0.000,B 0.000,C 90.000,E1 95.277} C_DIS
LIN {X 0.080,Y -485.070,Z 438.526,A 0.000,B 0.000,C 90.000,E1 94.759} C_DIS
LIN {X 0.060,Y -473.168,Z 438.518,A 0.000,B 0.000,C 90.000,E1 93.269} C_DIS
LIN {X 0.140,Y -455.694,Z 438.506,A 0.000,B 0.000,C 90.000,E1 90.974} C_DIS
LIN {X -0.161,Y -443.440,Z 438.495,A 0.000,B 0.000,C 90.000,E1 89.198} C_DIS
LIN {X 0.065,Y -428.490,Z 438.482,A 0.000,B 0.000,C 90.000,E1 86.788} C_DIS
LIN {X 0.016,Y -412.633,Z 438.467,A 0.000,B 0.000,C 90.000,E1 84.090} C_DIS
LIN {X -0.084,Y -400.320,Z 438.455,A 0.000,B 0.000,C 90.000,E1 81.894} C_DIS
LIN {X -0.071,Y -391.188,Z 438.446,A 0.000,B 0.000,C 90.000,E1 80.208} C_DIS
LIN {X -0.181,Y -380.601,Z 438.434,A 0.000,B 0.000,C 90.000,E1 78.229} C_DIS
LIN {X -0.012,Y -367.393,Z 438.420,A 0.000,B 0.000,C 90.000,E1 75.589} C_DIS
LIN {X 0.054,Y -352.373,Z 438.402,A 0.000,B 0.000,C 90.000,E1 72.308} C_DIS
LIN {X 0.067,Y -339.766,Z 438.385,A 0.000,B 0.000,C 90.000,E1 69.263} C_DIS
LIN {X 0.003,Y -330.159,Z 438.371,A 0.000,B 0.000,C 90.000,E1 66.794} C_DIS
LIN {X 0.044,Y -319.557,Z 438.355,A 0.000,B 0.000,C 90.000,E1 63.948} C_DIS
LIN {X 0.076,Y -309.324,Z 438.339,A 0.000,B 0.000,C 90.000,E1 61.051} C_DIS
LIN {X 0.025,Y -298.311,Z 438.321,A 0.000,B 0.000,C 90.000,E1 57.788} C_DIS
LIN {X -0.104,Y -288.225,Z 438.303,A 0.000,B 0.000,C 90.000,E1 54.482} C_DIS
LIN {X 0.047,Y -280.664,Z 438.288,A 0.000,B 0.000,C 90.000,E1 51.743} C_DIS
LIN {X -0.036,Y -274.896,Z 438.276,A 0.000,B 0.000,C 90.000,E1 49.703} C_DIS
LIN {X -0.084,Y -268.948,Z 438.265,A 0.000,B 0.000,C 90.000,E1 47.634} C_DIS
LIN {X 0.123,Y -262.748,Z 438.253,A 0.000,B 0.000,C 90.000,E1 45.486} C_DIS
LIN {X 0.022,Y -256.441,Z 438.241,A 0.000,B 0.000,C 90.000,E1 43.380} C_DIS
LIN {X 0.004,Y -249.985,Z 438.229,A 0.000,B 0.000,C 90.000,E1 41.229} C_DIS
LIN {X 0.036,Y -239.401,Z 438.209,A 0.000,B 0.000,C 90.000,E1 37.569} C_DIS
LIN {X -0.052,Y -231.535,Z 438.192,A 0.000,B 0.000,C 90.000,E1 34.612} C_DIS
LIN {X -0.076,Y -224.371,Z 438.175,A 0.000,B 0.000,C 90.000,E1 31.592} C_DIS
LIN {X 0.059,Y -218.037,Z 438.158,A 0.000,B 0.000,C 90.000,E1 28.487} C_DIS
LIN {X -0.076,Y -212.444,Z 438.141,A 0.000,B 0.000,C 90.000,E1 25.412} C_DIS
LIN {X -0.037,Y -206.416,Z 438.119,A 0.000,B 0.000,C 90.000,E1 21.461} C_DIS
LIN {X 0.014,Y -201.265,Z 438.097,A 0.000,B 0.000,C 90.000,E1 17.457} C_DIS
LIN {X 0.053,Y -197.143,Z 438.075,A 0.000,B 0.000,C 90.000,E1 13.411} C_DIS
LIN {X -0.069,Y -193.936,Z 438.052,A 0.000,B 0.000,C 90.000,E1 9.378} C_DIS
LIN {X 0.014,Y -191.069,Z 438.020,A 0.000,B 0.000,C 90.000,E1 3.612} C_DIS
LIN {X 0.048,Y -191.112,Z 437.965,A 0.000,B 0.000,C 90.000,E1 353.742} C_DIS
LIN {X 0.025,Y -193.977,Z 437.933,A 0.000,B 0.000,C 90.000,E1 347.993} C_DIS
LIN {X 0.047,Y -197.867,Z 437.906,A 0.000,B 0.000,C 90.000,E1 343.087} C_DIS
LIN {X 0.080,Y -202.142,Z 437.884,A 0.000,B 0.000,C 90.000,E1 339.028} C_DIS
LIN {X -0.026,Y -207.538,Z 437.861,A 0.000,B 0.000,C 90.000,E1 335.049} C_DIS
LIN {X 0.109,Y -213.758,Z 437.839,A 0.000,B 0.000,C 90.000,E1 331.051} C_DIS
LIN {X 0.018,Y -220.516,Z 437.818,A 0.000,B 0.000,C 90.000,E1 327.168} C_DIS
LIN {X -0.059,Y -227.951,Z 437.796,A 0.000,B 0.000,C 90.000,E1 323.336} C_DIS
LIN {X -0.043,Y -236.272,Z 437.775,A 0.000,B 0.000,C 90.000,E1 319.542} C_DIS
LIN {X 0.000,Y -244.638,Z 437.757,A 0.000,B 0.000,C 90.000,E1 316.176} C_DIS
LIN {X -0.047,Y -254.221,Z 437.738,A 0.000,B 0.000,C 90.000,E1 312.894} C_DIS
LIN {X 0.056,Y -265.010,Z 437.720,A 0.000,B 0.000,C 90.000,E1 309.644} C_DIS
LIN {X -0.030,Y -276.858,Z 437.703,A 0.000,B 0.000,C 90.000,E1 306.503} C_DIS
LIN {X -0.183,Y -288.111,Z 437.688,A 0.000,B 0.000,C 90.000,E1 303.785} C_DIS
LIN {X 0.054,Y -302.891,Z 437.669,A 0.000,B 0.000,C 90.000,E1 300.384} C_DIS
LIN {X 0.011,Y -318.956,Z 437.651,A 0.000,B 0.000,C 90.000,E1 297.129} C_DIS
LIN {X 0.056,Y -336.771,Z 437.633,A 0.000,B 0.000,C 90.000,E1 293.951} C_DIS
LIN {X 0.077,Y -352.892,Z 437.619,A 0.000,B 0.000,C 90.000,E1 291.482} C_DIS
LIN {X 0.140,Y -372.794,Z 437.604,A 0.000,B 0.000,C 90.000,E1 288.779} C_DIS
LIN {X -0.082,Y -394.524,Z 437.590,A 0.000,B 0.000,C 90.000,E1 286.205} C_DIS
LIN {X -0.180,Y -415.361,Z 437.578,A 0.000,B 0.000,C 90.000,E1 284.064} C_DIS
LIN {X 0.111,Y -428.342,Z 437.571,A 0.000,B 0.000,C 90.000,E1 282.771} C_DIS
LIN {X 0.172,Y -435.913,Z 437.567,A 0.000,B 0.000,C 90.000,E1 282.007} C_DIS
LIN {X -0.128,Y -445.698,Z 437.561,A 0.000,B 0.000,C 90.000,E1 281.007} C_DIS
LIN {X 0.049,Y -452.571,Z 437.557,A 0.000,B 0.000,C 90.000,E1 280.197} C_DIS
LIN {X -0.085,Y -458.977,Z 437.552,A 0.000,B 0.000,C 90.000,E1 279.434} C_DIS
LIN {X 0.220,Y -464.867,Z 437.548,A 0.000,B 0.000,C 90.000,E1 278.624} C_DIS
LIN {X -0.103,Y -471.892,Z 437.542,A 0.000,B 0.000,C 90.000,E1 277.644} C_DIS
LIN {X 0.127,Y -478.148,Z 437.537,A 0.000,B 0.000,C 90.000,E1 276.606} C_DIS
LIN {X 0.135,Y -482.348,Z 437.533,A 0.000,B 0.000,C 90.000,E1 275.853} C_DIS
LIN {X 0.133,Y -485.970,Z 437.528,A 0.000,B 0.000,C 90.000,E1 275.106} C_DIS
LIN {X -0.038,Y -487.026,Z 437.527,A 0.000,B 0.000,C 90.000,E1 274.878} C_DIS
LIN {X 0.161,Y -488.824,Z 437.524,A 0.000,B 0.000,C 90.000,E1 274.359} C_DIS
LIN {X -0.126,Y -490.230,Z 437.522,A 0.000,B 0.000,C 90.000,E1 273.898} C_DIS
LIN {X 0.056,Y -491.234,Z 437.519,A 0.000,B 0.000,C 90.000,E1 273.383} C_DIS
LIN {X -0.218,Y -491.821,Z 437.516,A 0.000,B 0.000,C 90.000,E1 272.922} C_DIS
LIN {X -0.018,Y -492.096,Z 437.513,A 0.000,B 0.000,C 90.000,E1 272.407} C_DIS
LIN {X 0.187,Y -491.967,Z 437.511,A 0.000,B 0.000,C 90.000,E1 271.892} C_DIS
LIN {X -0.084,Y -491.455,Z 437.508,A 0.000,B 0.000,C 90.000,E1 271.432} C_DIS
LIN {X 0.122,Y -490.508,Z 437.505,A 0.000,B 0.000,C 90.000,E1 270.917} C_DIS
LIN {X -0.164,Y -489.055,Z 437.502,A 0.000,B 0.000,C 90.000,E1 270.458} C_DIS
LIN {X 0.034,Y -487.101,Z 437.500,A 0.000,B 0.000,C 90.000,E1 269.943} C_DIS
LIN {X 0.222,Y -484.548,Z 437.497,A 0.000,B 0.000,C 90.000,E1 269.427} C_DIS
LIN {X -0.091,Y -481.302,Z 437.494,A 0.000,B 0.000,C 90.000,E1 268.969} C_DIS
LIN {X 0.059,Y -477.062,Z 437.491,A 0.000,B 0.000,C 90.000,E1 268.453} C_DIS
LIN {X -0.115,Y -474.585,Z 437.490,A 0.000,B 0.000,C 90.000,E1 268.224} C_DIS
LIN {X 0.207,Y -468.912,Z 437.487,A 0.000,B 0.000,C 90.000,E1 267.707} C_DIS
LIN {X 0.030,Y -462.543,Z 437.485,A 0.000,B 0.000,C 90.000,E1 267.306} C_DIS
LIN {X -0.057,Y -455.814,Z 437.483,A 0.000,B 0.000,C 90.000,E1 266.963} C_DIS
LIN {X -0.070,Y -448.886,Z 437.481,A 0.000,B 0.000,C 90.000,E1 266.674} C_DIS
LIN {X -0.169,Y -441.803,Z 437.480,A 0.000,B 0.000,C 90.000,E1 266.445} C_DIS
LIN {X 0.066,Y -434.266,Z 437.479,A 0.000,B 0.000,C 90.000,E1 266.216} C_DIS
LIN {X -0.186,Y -425.499,Z 437.478,A 0.000,B 0.000,C 90.000,E1 266.102} C_DIS
LIN {X -0.081,Y -414.825,Z 437.478,A 0.000,B 0.000,C 90.000,E1 265.988} C_DIS
LIN {X 0.141,Y -407.244,Z 437.477,A 0.000,B 0.000,C 90.000,E1 265.927} C_DIS
LIN {X 0.031,Y -180.918,Z 437.477,A 0.000,B 0.000,C 90.000,E1 265.927} C_DIS
LIN {X 0.064,Y -180.840,Z 437.472,A 0.000,B 0.000,C 90.000,E1 264.894} C_DIS
LIN {X -0.040,Y -178.881,Z 437.443,A 0.000,B 0.000,C 90.000,E1 259.690} C_DIS
LIN {X 0.036,Y -175.924,Z 437.414,A 0.000,B 0.000,C 90.000,E1 254.574} C_DIS
LIN {X -0.018,Y -175.362,Z 437.410,A 0.000,B 0.000,C 90.000,E1 253.740} C_DIS
LIN {X 0.040,Y -172.141,Z 437.386,A 0.000,B 0.000,C 90.000,E1 249.444} C_DIS
LIN {X 0.018,Y -171.605,Z 437.381,A 0.000,B 0.000,C 90.000,E1 248.592} C_DIS
LIN {X 0.006,Y -167.827,Z 437.357,A 0.000,B 0.000,C 90.000,E1 244.280} C_DIS
LIN {X 0.023,Y -166.552,Z 437.347,A 0.000,B 0.000,C 90.000,E1 242.538} C_DIS
LIN {X -0.066,Y -162.548,Z 437.323,A 0.000,B 0.000,C 90.000,E1 238.201} C_DIS
LIN {X -0.006,Y -161.226,Z 437.313,A 0.000,B 0.000,C 90.000,E1 236.421} C_DIS
LIN {X 0.030,Y -157.232,Z 437.289,A 0.000,B 0.000,C 90.000,E1 231.984} C_DIS
LIN {X 0.052,Y -155.956,Z 437.279,A 0.000,B 0.000,C 90.000,E1 230.194} C_DIS
LIN {X 0.010,Y -152.210,Z 437.254,A 0.000,B 0.000,C 90.000,E1 225.729} C_DIS
LIN {X 0.031,Y -150.454,Z 437.239,A 0.000,B 0.000,C 90.000,E1 223.014} C_DIS
LIN {X 0.058,Y -147.181,Z 437.214,A 0.000,B 0.000,C 90.000,E1 218.463} C_DIS
LIN {X 0.024,Y -145.198,Z 437.193,A 0.000,B 0.000,C 90.000,E1 214.818} C_DIS
LIN {X 0.059,Y -142.336,Z 437.163,A 0.000,B 0.000,C 90.000,E1 209.283} C_DIS
LIN {X -0.012,Y -141.725,Z 437.153,A 0.000,B 0.000,C 90.000,E1 207.462} C_DIS
LIN {X -0.029,Y -139.479,Z 437.116,A 0.000,B 0.000,C 90.000,E1 200.972} C_DIS
LIN {X -0.041,Y -138.978,Z 437.101,A 0.000,B 0.000,C 90.000,E1 198.181} C_DIS
LIN {X -0.056,Y -138.332,Z 437.054,A 0.000,B 0.000,C 90.000,E1 189.782} C_DIS
LIN {X -0.055,Y -139.431,Z 437.008,A 0.000,B 0.000,C 90.000,E1 181.375} C_DIS
LIN {X -0.002,Y -141.359,Z 436.971,A 0.000,B 0.000,C 90.000,E1 174.837} C_DIS
LIN {X -0.026,Y -142.712,Z 436.956,A 0.000,B 0.000,C 90.000,E1 172.064} C_DIS
LIN {X -0.067,Y -145.088,Z 436.930,A 0.000,B 0.000,C 90.000,E1 167.465} C_DIS
LIN {X 0.069,Y -147.713,Z 436.910,A 0.000,B 0.000,C 90.000,E1 163.740} C_DIS
LIN {X 0.011,Y -150.369,Z 436.890,A 0.000,B 0.000,C 90.000,E1 160.115} C_DIS
LIN {X 0.029,Y -153.796,Z 436.869,A 0.000,B 0.000,C 90.000,E1 156.485} C_DIS
LIN {X -0.051,Y -157.208,Z 436.849,A 0.000,B 0.000,C 90.000,E1 152.922} C_DIS
LIN {X 0.030,Y -161.372,Z 436.830,A 0.000,B 0.000,C 90.000,E1 149.331} C_DIS
LIN {X 0.042,Y -165.574,Z 436.810,A 0.000,B 0.000,C 90.000,E1 145.801} C_DIS
LIN {X 0.028,Y -170.493,Z 436.791,A 0.000,B 0.000,C 90.000,E1 142.316} C_DIS
LIN {X 0.073,Y -175.373,Z 436.772,A 0.000,B 0.000,C 90.000,E1 138.852} C_DIS
LIN {X -0.063,Y -180.998,Z 436.753,A 0.000,B 0.000,C 90.000,E1 135.486} C_DIS
LIN {X 0.061,Y -186.426,Z 436.734,A 0.000,B 0.000,C 90.000,E1 132.081} C_DIS
LIN {X 0.008,Y -191.052,Z 436.720,A 0.000,B 0.000,C 90.000,E1 129.600} C_DIS
LIN {X 0.024,Y -195.771,Z 436.705,A 0.000,B 0.000,C 90.000,E1 126.870} C_DIS
LIN {X -0.012,Y -294.631,Z 436.705,A 0.000,B 0.000,C 90.000,E1 126.870} C_DIS
LIN {X 0.009,Y -300.950,Z 436.703,A 0.000,B 0.000,C 90.000,E1 126.583} C_DIS
LIN {X 0.082,Y -303.801,Z 436.702,A 0.000,B 0.000,C 90.000,E1 126.297} C_DIS
LIN {X 0.044,Y -307.518,Z 436.699,A 0.000,B 0.000,C 90.000,E1 125.758} C_DIS
LIN {X -0.003,Y -309.088,Z 436.697,A 0.000,B 0.000,C 90.000,E1 125.438} C_DIS
LIN {X 0.064,Y -311.343,Z 436.693,A 0.000,B 0.000,C 90.000,E1 124.771} C_DIS
LIN {X 0.084,Y -322.162,Z 436.675,A 0.000,B 0.000,C 90.000,E1 121.544} C_DIS
LIN {X 0.099,Y -333.284,Z 436.659,A 0.000,B 0.000,C 90.000,E1 118.693} C_DIS
LIN {X -0.042,Y -345.818,Z 436.644,A 0.000,B 0.000,C 90.000,E1 115.924} C_DIS
LIN {X -0.186,Y -358.241,Z 436.630,A 0.000,B 0.000,C 90.000,E1 113.515} C_DIS
LIN {X 0.023,Y -371.961,Z 436.617,A 0.000,B 0.000,C 90.000,E1 111.099} C_DIS
LIN {X -0.036,Y -387.079,Z 436.604,A 0.000,B 0.000,C 90.000,E1 108.779} C_DIS
LIN {X 0.032,Y -403.705,Z 436.592,A 0.000,B 0.000,C 90.000,E1 106.496} C_DIS
LIN {X -0.104,Y -421.964,Z 436.579,A 0.000,B 0.000,C 90.000,E1 104.300} C_DIS
LIN {X -0.126,Y -441.733,Z 436.568,A 0.000,B 0.000,C 90.000,E1 102.175} C_DIS
LIN {X 0.025,Y -462.172,Z 436.557,A 0.000,B 0.000,C 90.000,E1 100.197} C_DIS
LIN {X 0.226,Y -485.610,Z 436.546,A 0.000,B 0.000,C 90.000,E1 98.163} C_DIS
LIN {X -0.126,Y -489.074,Z 436.543,A 0.000,B 0.000,C 90.000,E1 97.757} C_DIS
LIN {X 0.183,Y -490.344,Z 436.542,A 0.000,B 0.000,C 90.000,E1 97.473} C_DIS
LIN {X 0.071,Y -491.276,Z 436.540,A 0.000,B 0.000,C 90.000,E1 97.239} C_DIS
LIN {X -0.191,Y -492.283,Z 436.538,A 0.000,B 0.000,C 90.000,E1 96.777} C_DIS
LIN {X 0.041,Y -492.287,Z 436.535,A 0.000,B 0.000,C 90.000,E1 96.258} C_DIS
LIN {X -0.211,Y -491.287,Z 436.532,A 0.000,B 0.000,C 90.000,E1 95.796} C_DIS
LIN {X 0.127,Y -490.366,Z 436.531,A 0.000,B 0.000,C 90.000,E1 95.511} C_DIS
LIN {X 0.024,Y -489.106,Z 436.529,A 0.000,B 0.000,C 90.000,E1 95.277} C_DIS
LIN {X 0.244,Y -485.529,Z 436.527,A 0.000,B 0.000,C 90.000,E1 94.759} C_DIS
LIN {X -0.244,Y -473.643,Z 436.518,A 0.000,B 0.000,C 90.000,E1 93.326} C_DIS
LIN {X -0.142,Y -456.125,Z 436.506,A 0.000,B 0.000,C 90.000,E1 91.031} C_DIS
LIN {X 0.016,Y -443.822,Z 436.496,A 0.000,B 0.000,C 90.000,E1 89.198} C_DIS
LIN {X -0.182,Y -428.844,Z 436.482,A 0.000,B 0.000,C 90.000,E1 86.846} C_DIS
LIN {X -0.210,Y -412.974,Z 436.467,A 0.000,B 0.000,C 90.000,E1 84.147} C_DIS
LIN {X 0.103,Y -400.659,Z 436.455,A 0.000,B 0.000,C 90.000,E1 81.894} C_DIS
LIN {X 0.117,Y -391.538,Z 436.446,A 0.000,B 0.000,C 90.000,E1 80.208} C_DIS
LIN {X 0.009,Y -380.963,Z 436.435,A 0.000,B 0.000,C 90.000,E1 78.229} C_DIS
LIN {X -0.093,Y -366.343,Z 436.418,A 0.000,B 0.000,C 90.000,E1 75.338} C_DIS
LIN {X -0.113,Y -350.118,Z 436.399,A 0.000,B 0.000,C 90.000,E1 71.764} C_DIS
LIN {X -0.166,Y -338.840,Z 436.383,A 0.000,B 0.000,C 90.000,E1 69.028} C_DIS
LIN {X -0.124,Y -329.214,Z 436.370,A 0.000,B 0.000,C 90.000,E1 66.538} C_DIS
LIN {X -0.097,Y -318.631,Z 436.354,A 0.000,B 0.000,C 90.000,E1 63.691} C_DIS
LIN {X 0.008,Y -309.500,Z 436.339,A 0.000,B 0.000,C 90.000,E1 61.101} C_DIS
LIN {X -0.028,Y -298.452,Z 436.321,A 0.000,B 0.000,C 90.000,E1 57.837} C_DIS
LIN {X 0.094,Y -288.333,Z 436.303,A 0.000,B 0.000,C 90.000,E1 54.482} C_DIS
LIN {X 0.067,Y -280.772,Z 436.288,A 0.000,B 0.000,C 90.000,E1 51.778} C_DIS
LIN {X -0.054,Y -275.039,Z 436.276,A 0.000,B 0.000,C 90.000,E1 49.747} C_DIS
LIN {X 0.108,Y -269.097,Z 436.265,A 0.000,B 0.000,C 90.000,E1 47.634} C_DIS
LIN {X -0.060,Y -262.913,Z 436.253,A 0.000,B 0.000,C 90.000,E1 45.567} C_DIS
LIN {X 0.034,Y -256.616,Z 436.241,A 0.000,B 0.000,C 90.000,E1 43.419} C_DIS
LIN {X 0.002,Y -250.156,Z 436.229,A 0.000,B 0.000,C 90.000,E1 41.272} C_DIS
LIN {X 0.073,Y -239.583,Z 436.209,A 0.000,B 0.000,C 90.000,E1 37.604} C_DIS
LIN {X 0.131,Y -231.715,Z 436.192,A 0.000,B 0.000,C 90.000,E1 34.612} C_DIS
LIN {X 0.106,Y -224.540,Z 436.176,A 0.000,B 0.000,C 90.000,E1 31.592} C_DIS
LIN {X -0.057,Y -218.179,Z 436.159,A 0.000,B 0.000,C 90.000,E1 28.565} C_DIS
LIN {X -0.089,Y -212.560,Z 436.141,A 0.000,B 0.000,C 90.000,E1 25.463} C_DIS
LIN {X -0.127,Y -206.492,Z 436.119,A 0.000,B 0.000,C 90.000,E1 21.535} C_DIS
LIN {X -0.004,Y -201.303,Z 436.097,A 0.000,B 0.000,C 90.000,E1 17.511} C_DIS
LIN {X -0.013,Y -197.136,Z 436.075,A 0.000,B 0.000,C 90.000,E1 13.480} C_DIS
LIN {X 0.074,Y -193.381,Z 436.048,A 0.000,B 0.000,C 90.000,E1 8.568} C_DIS
LIN {X 0.039,Y -190.546,Z 436.011,A 0.000,B 0.000,C 90.000,E1 2.007} C_DIS
LIN {X -0.003,Y -191.296,Z 435.961,A 0.000,B 0.000,C 90.000,E1 352.932} C_DIS
LIN {X 0.018,Y -194.388,Z 435.929,A 0.000,B 0.000,C 90.000,E1 347.173} C_DIS
LIN {X -0.087,Y -198.501,Z 435.902,A 0.000,B 0.000,C 90.000,E1 342.308} C_DIS
LIN {X 0.032,Y -202.993,Z 435.879,A 0.000,B 0.000,C 90.000,E1 338.230} C_DIS
LIN {X 0.033,Y -208.565,Z 435.857,A 0.000,B 0.000,C 90.000,E1 334.229} C_DIS
LIN {X 0.008,Y -214.927,Z 435.835,A 0.000,B 0.000,C 90.000,E1 330.284} C_DIS
LIN {X 0.056,Y -221.825,Z 435.813,A 0.000,B 0.000,C 90.000,E1 326.373} C_DIS
LIN {X -0.038,Y -229.396,Z 435.792,A 0.000,B 0.000,C 90.000,E1 322.557} C_DIS
LIN {X -0.009,Y -237.920,Z 435.771,A 0.000,B 0.000,C 90.000,E1 318.771} C_DIS
LIN {X 0.088,Y -246.582,Z 435.752,A 0.000,B 0.000,C 90.000,E1 315.405} C_DIS
LIN {X -0.088,Y -255.266,Z 435.736,A 0.000,B 0.000,C 90.000,E1 312.528} C_DIS
LIN {X 0.047,Y -266.200,Z 435.718,A 0.000,B 0.000,C 90.000,E1 309.277} C_DIS
LIN {X -0.068,Y -279.548,Z 435.699,A 0.000,B 0.000,C 90.000,E1 305.804} C_DIS
LIN {X 0.118,Y -289.503,Z 435.686,A 0.000,B 0.000,C 90.000,E1 303.372} C_DIS
LIN {X -0.004,Y -304.406,Z 435.667,A 0.000,B 0.000,C 90.000,E1 300.050} C_DIS
LIN {X -0.004,Y -320.673,Z 435.649,A 0.000,B 0.000,C 90.000,E1 296.796} C_DIS
LIN {X -0.032,Y -336.794,Z 435.633,A 0.000,B 0.000,C 90.000,E1 293.951} C_DIS
LIN {X 0.115,Y -352.963,Z 435.619,A 0.000,B 0.000,C 90.000,E1 291.461} C_DIS
LIN {X -0.042,Y -370.613,Z 435.606,A 0.000,B 0.000,C 90.000,E1 289.087} C_DIS
